// SIMATIC STEP 7 (V5.x) project TEST_212
// station: _S7H_BUSSYSTEM_CT
// station: P_ADR_BUS
// station: Hardware
// station: ESTACION_01

SYMBOL_TABLE
"Z 1"	C 1	COUNTER
"Z 2"	C 2	COUNTER
"Z 3"	C 3	COUNTER
"Z 4"	C 4	COUNTER
"Z 5"	C 5	COUNTER
"Z 6"	C 6	COUNTER
"Z 7"	C 7	COUNTER
"Z 8"	C 8	COUNTER
"Z 9"	C 9	COUNTER
"Z 10"	C 10	COUNTER
"Z 11"	C 11	COUNTER
"Z 12"	C 12	COUNTER
"Z 13"	C 13	COUNTER
"Z 14"	C 14	COUNTER
"Z 15"	C 15	COUNTER
"Z 16"	C 16	COUNTER
"Z 17"	C 17	COUNTER
"Z 18"	C 18	COUNTER
"Z 19"	C 19	COUNTER
"Z 20"	C 20	COUNTER
"Z 21"	C 21	COUNTER
"Z 22"	C 22	COUNTER
"Z 23"	C 23	COUNTER
"Z 24"	C 24	COUNTER
"Z 25"	C 25	COUNTER
"Z 26"	C 26	COUNTER
"Z 27"	C 27	COUNTER
"Z 28"	C 28	COUNTER
"Z 29"	C 29	COUNTER
"Z 30"	C 30	COUNTER
"Z 31"	C 31	COUNTER
"Z 32"	C 32	COUNTER
"Z 33"	C 33	COUNTER
"Z 34"	C 34	COUNTER
"Z 35"	C 35	COUNTER
"Z 36"	C 36	COUNTER
"Z 37"	C 37	COUNTER
"Z 38"	C 38	COUNTER
"Z 39"	C 39	COUNTER
"Z 40"	C 40	COUNTER
"Z 41"	C 41	COUNTER
"Z 42"	C 42	COUNTER
"Z 43"	C 43	COUNTER
"Z 44"	C 44	COUNTER
"Z 45"	C 45	COUNTER
"Z 46"	C 46	COUNTER
"Z 47"	C 47	COUNTER
"Z 48"	C 48	COUNTER
"Z 49"	C 49	COUNTER
"Z 50"	C 50	COUNTER
"Z 51"	C 51	COUNTER
"Z 52"	C 52	COUNTER
"Z 53"	C 53	COUNTER
"Z 54"	C 54	COUNTER
"Z 55"	C 55	COUNTER
"Z 56"	C 56	COUNTER
"Z 57"	C 57	COUNTER
"Z 58"	C 58	COUNTER
"Z 59"	C 59	COUNTER
"Z 60"	C 60	COUNTER
"Z 61"	C 61	COUNTER
"Z 62"	C 62	COUNTER
"Z 63"	C 63	COUNTER
"Z 64"	C 64	COUNTER
"Z 65"	C 65	COUNTER
"Z 66"	C 66	COUNTER
"Z 67"	C 67	COUNTER
"Z 68"	C 68	COUNTER
"Z 69"	C 69	COUNTER
"Z 70"	C 70	COUNTER
"Z 71"	C 71	COUNTER
"Z 72"	C 72	COUNTER
"Z 73"	C 73	COUNTER
"Z 74"	C 74	COUNTER
"Z 75"	C 75	COUNTER
"Z 76"	C 76	COUNTER
"Z 77"	C 77	COUNTER
"Z 78"	C 78	COUNTER
"Z 79"	C 79	COUNTER
"Z 80"	C 80	COUNTER
"Z 81"	C 81	COUNTER
"Z 82"	C 82	COUNTER
"Z 83"	C 83	COUNTER
"Z 84"	C 84	COUNTER
"Z 85"	C 85	COUNTER
"Z 86"	C 86	COUNTER
"Z 87"	C 87	COUNTER
"Z 88"	C 88	COUNTER
"Z 89"	C 89	COUNTER
"Z 90"	C 90	COUNTER
"Z 91"	C 91	COUNTER
"Z 92"	C 92	COUNTER
"Z 93"	C 93	COUNTER
"Z 94"	C 94	COUNTER
"Z 95"	C 95	COUNTER
"Z 96"	C 96	COUNTER
"Z 97"	C 97	COUNTER
"Z 98"	C 98	COUNTER
"Z 99"	C 99	COUNTER
"Z 100"	C 100	COUNTER	// CONTADOR DE MINUTOS ( ALARMA  )
"Z 101"	C 101	COUNTER	// CONTADOR DE HORAS ( ALARMA  )
"Z 102"	C 102	COUNTER	// CONTADOR DE SEGUNDOS ( RELOJ  )
"Z 103"	C 103	COUNTER	// CONTADOR DE MINUTOS ( RELOJ )
"Z 104"	C 104	COUNTER	// CONTADOR DE HORAS ( RELOJ  )
"Z 105"	C 105	COUNTER	// CONTADOR DE RELOJ ( RELOJ DE 24 HORAS )
"Z 106"	C 106	COUNTER
"Z 107"	C 107	COUNTER
"Z 108"	C 108	COUNTER
"Z 109"	C 109	COUNTER
"Z 110"	C 110	COUNTER	// CONTADOR DE MINUTOS - AJUSTE DE ALARMAS
"Z 111"	C 111	COUNTER
"Z 112"	C 112	COUNTER
"Z 113"	C 113	COUNTER
"Z 114"	C 114	COUNTER
"Z 115"	C 115	COUNTER
"Z 116"	C 116	COUNTER
"Z 117"	C 117	COUNTER
"Z 118"	C 118	COUNTER
"Z 119"	C 119	COUNTER	// CONTADOR DE PERSONAS
"Z 120"	C 120	COUNTER	// CONTADOR ASCENDENTE / DESCENDENTE
"Z 121"	C 121	COUNTER	// CONTADOR ASCENDENTE
"Z 122"	C 122	COUNTER	// CONTADOR DESCENDENTE
"Z 123"	C 123	COUNTER
"Z 124"	C 124	COUNTER
"Z 125"	C 125	COUNTER
"Z 126"	C 126	COUNTER
"Z 127"	C 127	COUNTER	// CONTADOR DE IMPULSOS
"Z 128"	C 128	COUNTER
"Z 129"	C 129	COUNTER
"Z 130"	C 130	COUNTER
"Z 131"	C 131	COUNTER
"Z 132"	C 132	COUNTER
"Z 133"	C 133	COUNTER
"Z 134"	C 134	COUNTER
"Z 135"	C 135	COUNTER
"Z 136"	C 136	COUNTER
"Z 137"	C 137	COUNTER
"Z 138"	C 138	COUNTER
"Z 139"	C 139	COUNTER
"Z 140"	C 140	COUNTER
"Z 141"	C 141	COUNTER
"Z 142"	C 142	COUNTER
"Z 143"	C 143	COUNTER
"Z 144"	C 144	COUNTER
"Z 145"	C 145	COUNTER
"Z 146"	C 146	COUNTER
"Z 147"	C 147	COUNTER
"Z 148"	C 148	COUNTER
"Z 149"	C 149	COUNTER
"Z 150"	C 150	COUNTER
"Z 151"	C 151	COUNTER
"Z 152"	C 152	COUNTER
"Z 153"	C 153	COUNTER
"Z 154"	C 154	COUNTER
"Z 155"	C 155	COUNTER
"Z 156"	C 156	COUNTER
"Z 157"	C 157	COUNTER
"Z 158"	C 158	COUNTER
"Z 159"	C 159	COUNTER
"Z 160"	C 160	COUNTER
"Z 161"	C 161	COUNTER
"Z 162"	C 162	COUNTER
"Z 163"	C 163	COUNTER
"Z 164"	C 164	COUNTER
"Z 165"	C 165	COUNTER
"Z 166"	C 166	COUNTER
"Z 167"	C 167	COUNTER
"Z 168"	C 168	COUNTER
"Z 169"	C 169	COUNTER
"Z 170"	C 170	COUNTER
"Z 171"	C 171	COUNTER
"Z 172"	C 172	COUNTER
"Z 173"	C 173	COUNTER
"Z 174"	C 174	COUNTER
"Z 175"	C 175	COUNTER
"Z 176"	C 176	COUNTER
"Z 177"	C 177	COUNTER
"Z 178"	C 178	COUNTER
"Z 179"	C 179	COUNTER
"Z 180"	C 180	COUNTER
"Z 181"	C 181	COUNTER
"Z 182"	C 182	COUNTER
"Z 183"	C 183	COUNTER
"Z 184"	C 184	COUNTER
"Z 185"	C 185	COUNTER
"Z 186"	C 186	COUNTER
"Z 187"	C 187	COUNTER
"Z 188"	C 188	COUNTER
"Z 189"	C 189	COUNTER
"Z 190"	C 190	COUNTER
"Z 191"	C 191	COUNTER
"Z 192"	C 192	COUNTER
"Z 193"	C 193	COUNTER
"Z 194"	C 194	COUNTER
"Z 195"	C 195	COUNTER
"Z 196"	C 196	COUNTER
"Z 197"	C 197	COUNTER
"Z 198"	C 198	COUNTER
"Z 199"	C 199	COUNTER
"Z 200"	C 200	COUNTER
"Z 201"	C 201	COUNTER
"Z 202"	C 202	COUNTER
"Z 203"	C 203	COUNTER
"Z 204"	C 204	COUNTER
"Z 205"	C 205	COUNTER
"Z 206"	C 206	COUNTER
"Z 207"	C 207	COUNTER
"Z 208"	C 208	COUNTER
"Z 209"	C 209	COUNTER
"Z 210"	C 210	COUNTER
"Z 211"	C 211	COUNTER
"Z 212"	C 212	COUNTER
"Z 213"	C 213	COUNTER
"Z 214"	C 214	COUNTER
"Z 215"	C 215	COUNTER
"Z 216"	C 216	COUNTER
"Z 217"	C 217	COUNTER
"Z 218"	C 218	COUNTER
"Z 219"	C 219	COUNTER
"Z 220"	C 220	COUNTER
"Z 221"	C 221	COUNTER
"Z 222"	C 222	COUNTER
"Z 223"	C 223	COUNTER
"Z 224"	C 224	COUNTER
"Z 225"	C 225	COUNTER
"Z 226"	C 226	COUNTER
"Z 227"	C 227	COUNTER
"Z 228"	C 228	COUNTER
"Z 229"	C 229	COUNTER
"Z 230"	C 230	COUNTER
"Z 231"	C 231	COUNTER
"Z 232"	C 232	COUNTER
"Z 233"	C 233	COUNTER
"Z 234"	C 234	COUNTER
"Z 235"	C 235	COUNTER
"Z 236"	C 236	COUNTER
"Z 237"	C 237	COUNTER
"Z 238"	C 238	COUNTER
"Z 239"	C 239	COUNTER
"Z 240"	C 240	COUNTER
"Z 241"	C 241	COUNTER
"Z 242"	C 242	COUNTER
"Z 243"	C 243	COUNTER
"Z 244"	C 244	COUNTER
"Z 245"	C 245	COUNTER
"Z 246"	C 246	COUNTER
"Z 247"	C 247	COUNTER
"Z 248"	C 248	COUNTER
"Z 249"	C 249	COUNTER
"Z 250"	C 250	COUNTER
"Z 251"	C 251	COUNTER
"Z 252"	C 252	COUNTER
"Z 253"	C 253	COUNTER
"Z 254"	C 254	COUNTER
"Z 255"	C 255	COUNTER
"Z 256"	C 256	COUNTER
"DB 126"	DB 126	FB 126	// InstanzDB PNIODiag
"DB 127"	DB 127	DB 127	// InstanzDB STATDiag
"DB 208"	DB 208	DB 208	// DATOS GENERALES - TAK SIGNALE
"DB 228"	DB 228	DB 228	// SALVADO DE MARCAS OB35
"PNIODiag"	FB 126	FB 126	// Profibus/DP und Profinet/IO-Diagnose
"STATDiag"	FB 127	FB 127	// Zweitbaustein (PNIODiag)
"TE-M/V"	FC 10	FC 10	// FUNCIONAMIENTO DE ACCIONAMIENTO ( MOTOR / VALVULA )
"TE-SS"	FC 11	FC 11	// FUNCIONAMIENTO DE ACCIONAMIENTO ( VALVULA MOTORIZADA )
"TE-REK"	FC 12	FC 12	// FUNCIONAMIENTO DE ACCIONAMIENTO ( VALVULA DE CONTROL )
"TE-TS"	FC 13	FC 13	// FUNCIONAMIENTO DE ACCIONAMIENTO ( CONTROL PARCIAL )
"TE-VW3/3"	FC 14	FC 14	// FUNCIONAMIENTO DE ACCIONAMIENTO ( PRESELECCION 1 )
"TE-KO"	FC 15	FC 15	// FUNCIONAMIENTO DE CONTROL DE PASOS ( SECUENCIALES )
"TE-VW2/2"	FC 16	FC 16	// FUNCIONAMIENTO DE ACCIONAMIENTO ( PRESELECCION 1 )
"TE-VW2/1"	FC 17	FC 17	// FUNCIONAMIENTO DE ACCIONAMIENTO ( PRESELECCION 1 )
"TE_READ_RTM"	FC 18	FC 18	// TIEMPO DE FUNCIONAMIENTO DE UN ACCIONAMIENTO
"TE-WL ( PEA )"	FC 20	FC 20	// SENTRON WL ( IMAGEN DE PROCESO DE SALIDAS )
"TE-WL ( PEE )"	FC 25	FC 25	// SENTRON WL ( IMAGEN DE PROCESO DE ENTRADAS )
"TE-TAK"	FC 29	FC 29	// FUNCION DE GENERACION DE IMPULSOS
"TE-GRENZ"	FC 36	FC 36	// FUNCION DE LIMITE DE ALARMAS
"TE-RETTEN"	FC 38	FC 38	// SALVADO DE MARCAS DE TRABAJO
"TE-LADEN"	FC 39	FC 39	// CARGA DE MARCAS DE TRABAJO
"TE-SCHALTER"	FC 49	FC 49	// ANALOGSCHALTER - FUNKTION
"G7_STD_3"	FC 72	FC 72	// CONTROL DE OPERACION DE SECUENCIAS - GRAPH 7
"TE-ANEI"	FC 78	FC 78	// FUNCION DE LECTURA ANALOGICA
"TE-ANAU"	FC 79	FC 79	// FUNCION DE SALIDA ANALOGICA
"FC 110"	FC 110	FC 110	// FUNCIONES BASICAS
"FC 111"	FC 111	FC 111	// OPERACIONES LOGICAS BINARIAS
"FC 112"	FC 112	FC 112	// FUNCIONES DE MEMORIA
"FC 113"	FC 113	FC 113	// TEMPORIZADORES
"FC 114"	FC 114	FC 114	// CONTADORES
"FC 120"	FC 120	FC 120	// EJEMPLOS DE LAS FUNCIONES BINARIAS
"FC 121"	FC 121	FC 121	// SUPERVISION DE VENTILADORES
"FC 122"	FC 122	FC 122	// SUPERVISION DE FRECUENCIAS
"FC 123"	FC 123	FC 123	// CONTADOR DE PERSONAL
"FC 124"	FC 124	FC 124	// GENERADOR DE IMPULSOS
"FC 125"	FC 125	FC 125	// SEMAFORO
"FC 130"	FC 130	FC 130	// DIAGRAMAS ELECTRICOS
"FC 131"	FC 131	FC 131	// EJERCICIO No. 1 - CIRCUITO DE ENCLAVAMIENTO
"FC 132"	FC 132	FC 132	// EJERCICIO No. 2 - CIRCUITO DE TEMPORIZACION
"FC 133"	FC 133	FC 133	// EJERCICIO No. 3 - INVERSION DE GIRO
"FC 134"	FC 134	FC 134	// EJERCICIO No. 4 - ARRANQUE ESTRELLA - TRIANGULO
"FC 135"	FC 135	FC 135	// EJERCICIO No. 5 - INVERSION DE GIRO CON ARRANQUE ESTRELLA  - TRIANGULO
"FC 136"	FC 136	FC 136	// EJERCICIO No. 6 - CONEXION DAHLANDER
"FC 137"	FC 137	FC 137	// EJERCICIO No. 7 - MONTACARGAS
"FC 140"	FC 140	FC 140	// EJERCICIOS DE FUNCIONES BINARIAS
"FC 141"	FC 141	FC 141	// EJERCICIO No. 1 - SEMAFORO
"FC 142"	FC 142	FC 142	// EJERCICIO No. 2 - RELOJ DESPERTADOR
"FC 143"	FC 143	FC 143	// EJERCICIO No. 3 - PANEL DE ALARMAS
"FC 144"	FC 144	FC 144	// EJERCICIO No. 4 - ARRANQUE Y PARO DE MOTORES
"FC 145"	FC 145	FC 145	// EJERCICIO No. 5 - ELEVADOR
"FC 150"	FC 150	FC 150
"FC 151"	FC 151	FC 151
"FC 160"	FC 160	FC 160	// DIAGRAMAS ELECTRONEUMATICOS
"FC 161"	FC 161	FC 161	// EJERCICIO No. 1 -
"FC 162"	FC 162	FC 162	// EJERCICIO No. 2 -
"FC 163"	FC 163	FC 163	// EJERCICIO No. 3 -
"FC 164"	FC 164	FC 164	// EJERCICIO No. 4 -
"FC 165"	FC 165	FC 165	// EJERCICIO No. 5 -
"FC 166"	FC 166	FC 166	// EJERCICIO No. 6 -
"FC 167"	FC 167	FC 167	// EJERCICIO No. 7 -
"FC 240"	FC 240	FC 240	// INDICACION DE ESTADO - PANEL DE OPERACION
"FC 248"	FC 248	FC 248	// INDICACION DE CONTACTORES
"FC 249"	FC 249	FC 249	// INDICACION DE SELECTORES
"FC 250"	FC 250	FC 250	// SIMULACION DE RETROAVISOS
"FC 251"	FC 251	FC 251	// SIMULACION DE RETROAVISOS # 1
"FC 252"	FC 252	FC 252	// SIMULACION DE RETROAVISOS # 2
"FC 253"	FC 253	FC 253	// SIMULACION DE RETROAVISOS # 3
"FC 254"	FC 254	FC 254	// SIMULACION DE RETROAVISOS # 4
"FC 255"	FC 255	FC 255	// SIMULACION DE RETROAVISOS # 5
"FC 256"	FC 256	FC 256	// SIMULACION DE RETROAVISOS # 6
"FC 257"	FC 257	FC 257	// SIMULACION DE RETROAVISOS # 7
"1S2"	I 0.0	BOOL	// BOTON PULSADOR DE ARRANQUE # 1
"2S2"	I 0.1	BOOL	// BOTON PULSADOR DE ARRANQUE # 2
"3S2"	I 0.2	BOOL	// BOTON PULSADOR DE ARRANQUE # 3
"4S2"	I 0.3	BOOL	// BOTON PULSADOR DE ARRANQUE # 4
"5S2"	I 0.4	BOOL	// BOTON PULSADOR DE ARRANQUE # 5
"6S2"	I 0.5	BOOL	// BOTON PULSADOR DE ARRANQUE # 6
"7S2"	I 0.6	BOOL	// BOTON PULSADOR DE ARRANQUE # 7
"8S2"	I 0.7	BOOL	// BOTON PULSADOR DE ARRANQUE # 8
"1S3"	I 1.0	BOOL	// BOTON PULSADOR DE PARO # 1
"2S3"	I 1.1	BOOL	// BOTON PULSADOR DE PARO # 2
"3S3"	I 1.2	BOOL	// BOTON PULSADOR DE PARO # 3
"4S3"	I 1.3	BOOL	// BOTON PULSADOR DE PARO # 4
"5S3"	I 1.4	BOOL	// BOTON PULSADOR DE PARO # 5
"6S3"	I 1.5	BOOL	// BOTON PULSADOR DE PARO # 6
"7S3"	I 1.6	BOOL	// BOTON PULSADOR DE PARO # 7
"8S3"	I 1.7	BOOL	// BOTON PULSADOR DE PARO # 8
"1FR1"	I 2.0	BOOL	// DISPOSITIVO DE PROTECCION ( POR UMBRAL DE INTENSIDAD ) # 1
"2FR1"	I 2.1	BOOL	// DISPOSITIVO DE PROTECCION ( POR UMBRAL DE INTENSIDAD ) # 2
"3FR1"	I 2.2	BOOL	// DISPOSITIVO DE PROTECCION ( POR UMBRAL DE INTENSIDAD ) # 3
"4FR1"	I 2.3	BOOL	// DISPOSITIVO DE PROTECCION ( POR UMBRAL DE INTENSIDAD ) # 4
"5FR1"	I 2.4	BOOL	// DISPOSITIVO DE PROTECCION ( POR UMBRAL DE INTENSIDAD ) # 5
"6FR1"	I 2.5	BOOL	// DISPOSITIVO DE PROTECCION ( POR UMBRAL DE INTENSIDAD ) # 6
"7FR1"	I 2.6	BOOL	// DISPOSITIVO DE PROTECCION ( POR UMBRAL DE INTENSIDAD ) # 7
"8FR1"	I 2.7	BOOL	// DISPOSITIVO DE PROTECCION ( POR UMBRAL DE INTENSIDAD ) # 8
"E 3.0"	I 3.0	BOOL
"E 3.1"	I 3.1	BOOL
"E 3.2"	I 3.2	BOOL
"E 3.3"	I 3.3	BOOL
"E 3.4"	I 3.4	BOOL
"E 3.5"	I 3.5	BOOL
"E 3.6"	I 3.6	BOOL
"E 3.7"	I 3.7	BOOL
"5KM1_12"	I 4.0	BOOL	// CONTACTOR PRINCIPAL - 5KM1 ( DESCONECTADO )
"5KM1_14"	I 4.1	BOOL	// CONTACTOR PRINCIPAL - 5KM1 ( CONECTADO )
"5KM2_12"	I 4.2	BOOL	// CONTACTOR PRINCIPAL - 5KM2 ( DESCONECTADO )
"5KM2_14"	I 4.3	BOOL	// CONTACTOR PRINCIPAL - 5KM2 ( CONECTADO )
"5KM3_12"	I 4.4	BOOL	// CONTACTOR PRINCIPAL - 5KM3 ( DESCONECTADO )
"5KM3_14"	I 4.5	BOOL	// CONTACTOR PRINCIPAL - 5KM3 ( CONECTADO )
"5KM4_12"	I 4.6	BOOL	// CONTACTOR PRINCIPAL - 5KM4 ( DESCONECTADO )
"5KM4_14"	I 4.7	BOOL	// CONTACTOR PRINCIPAL - 5KM4 ( CONECTADO )
"6KM1_12"	I 5.0	BOOL	// CONTACTOR PRINCIPAL - 6KM1 ( DESCONECTADO )
"6KM1_14"	I 5.1	BOOL	// CONTACTOR PRINCIPAL - 6KM1 ( CONECTADO )
"6KM2_12"	I 5.2	BOOL	// CONTACTOR PRINCIPAL - 6KM2 ( DESCONECTADO )
"6KM2_14"	I 5.3	BOOL	// CONTACTOR PRINCIPAL - 6KM2 ( CONECTADO )
"6KM3_12"	I 5.4	BOOL	// CONTACTOR PRINCIPAL - 6KM3 ( DESCONECTADO )
"6KM3_14"	I 5.5	BOOL	// CONTACTOR PRINCIPAL - 6KM3 ( CONECTADO )
"E 5.6"	I 5.6	BOOL
"E 5.7"	I 5.7	BOOL
"1KM1_12"	I 6.0	BOOL	// CONTACTOR PRINCIPAL - 1KM1 ( DESCONECTADO )
"1KM1_14"	I 6.1	BOOL	// CONTACTOR PRINCIPAL - 1KM1 ( CONECTADO )
"2KM1_12"	I 6.2	BOOL	// CONTACTOR PRINCIPAL - 2KM1 ( DESCONECTADO )
"2KM1_14"	I 6.3	BOOL	// CONTACTOR PRINCIPAL - 2KM1 ( CONECTADO )
"2KM2_12"	I 6.4	BOOL	// CONTACTOR PRINCIPAL - 2KM2 ( DESCONECTADO )
"2KM2_14"	I 6.5	BOOL	// CONTACTOR PRINCIPAL - 2KM2 ( CONECTADO )
"E 6.6"	I 6.6	BOOL
"E 6.7"	I 6.7	BOOL
"BE4"	I 8.0	BOOL	// TRANSPORTADOR - SENSOR LB
"S1"	I 8.1	BOOL	// TRANSPORTADOR - BOTON PULSADOR T_BAY1
"S2"	I 8.2	BOOL	// TRANSPORTADOR - BOTON PULSADOR T_BAY2
"S3"	I 8.3	BOOL	// TRANSPORTADOR - BOTON PULSADOR T_BAY3
"S4"	I 8.4	BOOL	// TRANSPORTADOR - BOTON PULSADOR T_BAY-LB
"BE1"	I 8.5	BOOL	// TRANSPORTADOR - SENSOR BAY1
"BE2"	I 8.6	BOOL	// TRANSPORTADOR - SENSOR BAY2
"BE3"	I 8.7	BOOL	// TRANSPORTADOR - SENSOR BAY3
"3KM1_12"	I 12.0	BOOL	// CONTACTOR PRINCIPAL - 3KM1 ( DESCONECTADO )
"3KM1_14"	I 12.1	BOOL	// CONTACTOR PRINCIPAL - 3KM1 ( CONECTADO )
"3KM2_12"	I 12.2	BOOL	// CONTACTOR PRINCIPAL - 3KM2 ( DESCONECTADO )
"3KM2_14"	I 12.3	BOOL	// CONTACTOR PRINCIPAL - 3KM2 ( CONECTADO )
"E 12.4"	I 12.4	BOOL
"E 12.5"	I 12.5	BOOL
"E 12.6"	I 12.6	BOOL
"E 12.7"	I 12.7	BOOL
"4KM1_12"	I 13.0	BOOL	// CONTACTOR PRINCIPAL - 4KM1 ( DESCONECTADO )
"4KM1_14"	I 13.1	BOOL	// CONTACTOR PRINCIPAL - 4KM1 ( CONECTADO )
"4KM2_12"	I 13.2	BOOL	// CONTACTOR PRINCIPAL - 4KM2 ( DESCONECTADO )
"4KM2_14"	I 13.3	BOOL	// CONTACTOR PRINCIPAL - 4KM2 ( CONECTADO )
"4KM3_12"	I 13.4	BOOL	// CONTACTOR PRINCIPAL - 4KM3 ( DESCONECTADO )
"4KM3_14"	I 13.5	BOOL	// CONTACTOR PRINCIPAL - 4KM3 ( CONECTADO )
"E 13.6"	I 13.6	BOOL
"E 13.7"	I 13.7	BOOL
"E 14.0"	I 14.0	BOOL
"E 14.1"	I 14.1	BOOL
"E 14.2"	I 14.2	BOOL
"E 14.3"	I 14.3	BOOL
"E 14.4"	I 14.4	BOOL
"E 14.5"	I 14.5	BOOL
"E 14.6"	I 14.6	BOOL
"E 14.7"	I 14.7	BOOL
"E 15.0"	I 15.0	BOOL
"E 15.1"	I 15.1	BOOL
"E 15.2"	I 15.2	BOOL
"E 15.3"	I 15.3	BOOL
"E 15.4"	I 15.4	BOOL
"E 15.5"	I 15.5	BOOL
"E 15.6"	I 15.6	BOOL
"E 15.7"	I 15.7	BOOL
"7KM1_12"	I 16.0	BOOL	// CONTACTOR DE VELOCIDAD LENTA ( DESCONECTADO )
"7KM1_14"	I 16.1	BOOL
"7KM2_12"	I 16.2	BOOL	// CONTACTOR DE VELOCIDAD RAPIDA ( DESCONECTADO )
"7KM2_!4"	I 16.3	BOOL
"7KM3_12"	I 16.4	BOOL	// CONTACTOR DE VELOCIDAD RAPIDA ( DESCONECTADO )
"7KM3_14"	I 16.5	BOOL	// CONTACTOR DE VELOCIDAD RAPIDA ( CONECTADO )
"7QS10"	I 16.6	BOOL	// DETECTOR DE PLANTA BAJA
"7QS20"	I 16.7	BOOL	// DETECTOR PRIMER PISO
"7KM10_12"	I 17.0	BOOL	// CONTACTOR DE BAJADA ( DESCONECTADO )
"7KM10_14"	I 17.1	BOOL	// CONTACTOR DE BAJADA ( CONECTADO )
"7KM20_12"	I 17.2	BOOL	// CONTACTOR DE SUBIDA ( DESCONECTADO )
"7KM20_14"	I 17.3	BOOL	// CONTACTOR DE SUBIDA ( CONECTADO )
"7SB1"	I 17.4	BOOL	// COMANDO DE LLAMADA A PLANTA BAJA
"7SB2"	I 17.5	BOOL	// COMANDO DE LLAMADA A PRIMER PISO
"7SB3"	I 17.6	BOOL	// COMANDO DE PARO
"1S1A"	I 124.0	BOOL	// POSICION LOCAL - SELECTOR # 1
"1S1B"	I 124.1	BOOL	// POSICION REMOTO - SELECTOR # 1
"2S1A"	I 124.2	BOOL	// POSICION LOCAL - SELECTOR # 2
"2S1B"	I 124.3	BOOL	// POSICION REMOTO - SELECTOR # 2
"3S1A"	I 124.4	BOOL	// POSICION LOCAL - SELECTOR # 3
"3S1B"	I 124.5	BOOL	// POSICION REMOTO - SELECTOR # 3
"4S1A"	I 124.6	BOOL	// POSICION LOCAL - SELECTOR # 4
"4S1B"	I 124.7	BOOL	// POSICION REMOTO - SELECTOR # 4
"5S1A"	I 125.0	BOOL	// POSICION LOCAL - SELECTOR # 5
"5S1B"	I 125.1	BOOL	// POSICION REMOTO - SELECTOR # 5
"6S1A"	I 125.2	BOOL	// POSICION LOCAL - SELECTOR # 6
"6S1B"	I 125.3	BOOL	// POSICION REMOTO - SELECTOR # 6
"7S1A"	I 125.4	BOOL	// POSICION LOCAL - SELECTOR # 7
"7S1B"	I 125.5	BOOL	// POSICION REMOTO - SELECTOR # 7
"8S1A"	I 125.6	BOOL	// POSICION LOCAL - SELECTOR # 8
"8S1B"	I 125.7	BOOL	// POSICION REMOTO - SELECTOR # 8
"´0´"	M 0.0	BOOL	// CERO LOGICO
"´1´"	M 0.1	BOOL	// UNO LOGICO
"M 0.2"	M 0.2	BOOL
"M 0.3"	M 0.3	BOOL
"M 0.4"	M 0.4	BOOL
"M 0.5"	M 0.5	BOOL
"M 0.6"	M 0.6	BOOL	// MARCA DE INICIO - PROGRAMA DE TIEMPO ( 100 ms )
"M 0.7"	M 0.7	BOOL	// MARCA DE INICIO - EJECUCION CICLICA DE PROGRAMA
"M 1.0"	M 1.0	BOOL
"M 1.1"	M 1.1	BOOL
"M 1.2"	M 1.2	BOOL	// FLANCO 0.5 Seg.
"M 1.3"	M 1.3	BOOL	// FLANCO 1.0 Seg.
"M 1.4"	M 1.4	BOOL	// FLANCO 2.0 Seg.
"M 1.5"	M 1.5	BOOL	// PULSOS 0.5 Seg.
"M 1.6"	M 1.6	BOOL	// PULSOS 1.0 Seg.
"M 1.7"	M 1.7	BOOL	// PULSOS 2.0 Seg.
"M 2.0"	M 2.0	BOOL
"M 2.1"	M 2.1	BOOL
"M 2.2"	M 2.2	BOOL
"M 2.3"	M 2.3	BOOL
"M 2.4"	M 2.4	BOOL
"M 2.5"	M 2.5	BOOL
"M 2.6"	M 2.6	BOOL
"M 2.7"	M 2.7	BOOL
"M 3.0"	M 3.0	BOOL
"M 3.1"	M 3.1	BOOL
"M 3.2"	M 3.2	BOOL
"M 3.3"	M 3.3	BOOL
"M 3.4"	M 3.4	BOOL
"M 3.5"	M 3.5	BOOL
"M 3.6"	M 3.6	BOOL
"M 3.7"	M 3.7	BOOL
"M 4.0"	M 4.0	BOOL
"M 4.1"	M 4.1	BOOL
"M 4.2"	M 4.2	BOOL
"M 4.3"	M 4.3	BOOL
"M 4.4"	M 4.4	BOOL
"M 4.5"	M 4.5	BOOL
"M 4.6"	M 4.6	BOOL
"M 4.7"	M 4.7	BOOL
"M 5.0"	M 5.0	BOOL
"M 5.1"	M 5.1	BOOL
"M 5.2"	M 5.2	BOOL
"M 5.3"	M 5.3	BOOL
"M 5.4"	M 5.4	BOOL
"M 5.5"	M 5.5	BOOL
"M 5.6"	M 5.6	BOOL
"M 5.7"	M 5.7	BOOL
"M 6.0"	M 6.0	BOOL
"M 6.1"	M 6.1	BOOL
"M 6.2"	M 6.2	BOOL
"M 6.3"	M 6.3	BOOL
"M 6.4"	M 6.4	BOOL
"M 6.5"	M 6.5	BOOL
"M 6.6"	M 6.6	BOOL
"M 6.7"	M 6.7	BOOL
"M 7.0"	M 7.0	BOOL
"M 7.1"	M 7.1	BOOL
"M 7.2"	M 7.2	BOOL
"M 7.3"	M 7.3	BOOL
"M 7.4"	M 7.4	BOOL
"M 7.5"	M 7.5	BOOL
"M 7.6"	M 7.6	BOOL
"M 7.7"	M 7.7	BOOL
"M 8.0"	M 8.0	BOOL
"M 8.1"	M 8.1	BOOL
"M 8.2"	M 8.2	BOOL
"M 8.3"	M 8.3	BOOL
"M 8.4"	M 8.4	BOOL
"M 8.5"	M 8.5	BOOL
"M 8.6"	M 8.6	BOOL
"M 8.7"	M 8.7	BOOL
"M 9.0"	M 9.0	BOOL
"M 9.1"	M 9.1	BOOL
"M 9.2"	M 9.2	BOOL
"M 9.3"	M 9.3	BOOL
"M 9.4"	M 9.4	BOOL
"M 9.5"	M 9.5	BOOL
"M 9.6"	M 9.6	BOOL
"M 9.7"	M 9.7	BOOL
"M 10.0"	M 10.0	BOOL	// PANEL DE OPERACION ( COMANDO DE ARRANQUE )
"M 10.7"	M 10.7	BOOL	// MARCA AUXILIAR - COMANDO DE ARRANQUE
"M 11.0"	M 11.0	BOOL	// PANEL DE OPERACION ( BOTON PULSADOR DE  ARRANQUE # 1 )
"M 11.1"	M 11.1	BOOL	// PANEL DE OPERACION ( BOTON PULSADOR DE  ARRANQUE # 2 )
"M 11.2"	M 11.2	BOOL	// PANEL DE OPERACION ( BOTON PULSADOR DE PARO )
"M 11.3"	M 11.3	BOOL
"M 11.4"	M 11.4	BOOL	// MARCA AUXILIAR - SIMULACION DE RETROAVISOS # 1
"M 11.5"	M 11.5	BOOL	// MARCA AUXILIAR - COMANDO DE PARO
"M 11.6"	M 11.6	BOOL	// MARCA AUXILIAR - COMANDO DE ARRANQUE # 2
"M 11.7"	M 11.7	BOOL	// MARCA AUXILIAR - COMANDO DE ARRANQUE # 1
"M 12.0"	M 12.0	BOOL	// PANEL DE OPERACION ( BOTON PULSADOR DE  ARRANQUE # 1 )
"M 12.1"	M 12.1	BOOL	// PANEL DE OPERACION ( BOTON PULSADOR DE  ARRANQUE # 2 )
"M 12.2"	M 12.2	BOOL	// PANEL DE OPERACION ( BOTON PULSADOR DE PARO )
"M 12.3"	M 12.3	BOOL	// MARCA AUXILIAR - SIMULACION DE RETROAVISOS # 2
"M 12.4"	M 12.4	BOOL	// MARCA AUXILIAR - SIMULACION DE RETROAVISOS # 1
"M 12.5"	M 12.5	BOOL	// MARCA AUXILIAR - COMANDO DE PARO
"M 12.6"	M 12.6	BOOL	// MARCA AUXILIAR - COMANDO DE ARRANQUE # 2
"M 12.7"	M 12.7	BOOL	// MARCA AUXILIAR - COMANDO DE ARRANQUE # 1
"M 13.0"	M 13.0	BOOL	// PANEL DE OPERACION ( BOTON PULSADOR DE  ARRANQUE # 1 )
"M 13.1"	M 13.1	BOOL	// PANEL DE OPERACION ( BOTON PULSADOR DE  ARRANQUE # 2 )
"M 13.2"	M 13.2	BOOL	// PANEL DE OPERACION ( BOTON PULSADOR DE PARO )
"M 13.3"	M 13.3	BOOL	// MARCA AUXILIAR - SIMULACION DE RETROAVISOS # 2
"M 13.4"	M 13.4	BOOL	// MARCA AUXILIAR - SIMULACION DE RETROAVISOS # 1
"M 13.5"	M 13.5	BOOL	// MARCA AUXILIAR - COMANDO DE PARO
"M 13.6"	M 13.6	BOOL	// MARCA AUXILIAR - COMANDO DE ARRANQUE # 2
"M 13.7"	M 13.7	BOOL	// MARCA AUXILIAR - COMANDO DE ARRANQUE # 1
"M 14.0"	M 14.0	BOOL	// PANEL DE OPERACION ( BOTON PULSADOR DE  ARRANQUE # 1 )
"M 14.1"	M 14.1	BOOL	// PANEL DE OPERACION ( BOTON PULSADOR DE  ARRANQUE # 2 )
"M 14.2"	M 14.2	BOOL	// PANEL DE OPERACION ( BOTON PULSADOR DE PARO )
"M 14.3"	M 14.3	BOOL	// MARCA AUXILIAR - SIMULACION DE RETROAVISOS # 2
"M 14.4"	M 14.4	BOOL	// MARCA AUXILIAR - SIMULACION DE RETROAVISOS # 1
"M 14.5"	M 14.5	BOOL	// MARCA AUXILIAR - COMANDO DE PARO
"M 14.6"	M 14.6	BOOL	// MARCA AUXILIAR - COMANDO DE ARRANQUE # 2
"M 14.7"	M 14.7	BOOL	// MARCA AUXILIAR - COMANDO DE ARRANQUE # 1
"M 15.0"	M 15.0	BOOL	// PANEL DE OPERACION ( BOTON PULSADOR DE  ARRANQUE # 1 )
"M 15.1"	M 15.1	BOOL	// PANEL DE OPERACION ( BOTON PULSADOR DE  ARRANQUE # 2 )
"M 15.2"	M 15.2	BOOL	// PANEL DE OPERACION ( BOTON PULSADOR DE PARO )
"M 15.3"	M 15.3	BOOL	// MARCA AUXILIAR - SIMULACION DE RETROAVISOS # 2
"M 15.4"	M 15.4	BOOL	// MARCA AUXILIAR - SIMULACION DE RETROAVISOS # 1
"M 15.5"	M 15.5	BOOL	// MARCA AUXILIAR - COMANDO DE PARO
"M 15.6"	M 15.6	BOOL	// MARCA AUXILIAR - COMANDO DE ARRANQUE # 2
"M 15.7"	M 15.7	BOOL	// MARCA AUXILIAR - COMANDO DE ARRANQUE # 1
"M 16.0"	M 16.0	BOOL	// PANEL DE OPERACION ( BOTON PULSADOR DE  ARRANQUE # 1 )
"M 16.1"	M 16.1	BOOL	// PANEL DE OPERACION ( BOTON PULSADOR DE  ARRANQUE # 2 )
"M 16.2"	M 16.2	BOOL	// PANEL DE OPERACION ( BOTON PULSADOR DE PARO )
"M 16.3"	M 16.3	BOOL	// MARCA AUXILIAR - SIMULACION DE RETROAVISOS # 2
"M 16.4"	M 16.4	BOOL	// MARCA AUXILIAR - SIMULACION DE RETROAVISOS # 1
"M 16.5"	M 16.5	BOOL	// MARCA AUXILIAR - COMANDO DE PARO
"M 16.6"	M 16.6	BOOL	// MARCA AUXILIAR - COMANDO DE ARRANQUE # 2
"M 16.7"	M 16.7	BOOL	// MARCA AUXILIAR - COMANDO DE ARRANQUE # 1
"M 17.0"	M 17.0	BOOL	// PANEL DE OPERACION ( COMANDO - LLAMADA A PLANTA BAJA  )
"M 17.1"	M 17.1	BOOL	// PANEL DE OPERACION ( COMANDO - LLAMADA A PRIMER PISO  )
"M 17.2"	M 17.2	BOOL	// PANEL DE OPERACION ( COMANDO DE PARO - MONTACARGAS )
"M 17.3"	M 17.3	BOOL	// MARCA AUXILIAR - SIMULACION DE RETROAVISOS # 2
"M 17.4"	M 17.4	BOOL	// MARCA AUXILIAR - SIMULACION DE RETROAVISOS # 1
"M 17.5"	M 17.5	BOOL	// MARCA AUXILIAR - COMANDO DE PARO
"M 17.6"	M 17.6	BOOL	// MARCA AUXILIAR - COMANDO DE ARRANQUE # 2
"M 17.7"	M 17.7	BOOL	// MARCA AUXILIAR - COMANDO DE ARRANQUE # 1
"M 18.0"	M 18.0	BOOL
"M 18.1"	M 18.1	BOOL
"M 18.2"	M 18.2	BOOL
"M 18.3"	M 18.3	BOOL	// MARCA AUXILIAR - SIMULACION DE RETROAVISOS # 4
"M 18.4"	M 18.4	BOOL	// MARCA AUXILIAR - SIMULACION DE RETROAVISOS # 3
"M 18.5"	M 18.5	BOOL
"M 18.6"	M 18.6	BOOL
"M 18.7"	M 18.7	BOOL
"M 19.0"	M 19.0	BOOL
"M 19.1"	M 19.1	BOOL
"M 19.2"	M 19.2	BOOL
"M 19.3"	M 19.3	BOOL	// MARCA AUXILIAR - SIMULACION DE RETROAVISOS # 3
"M 19.4"	M 19.4	BOOL	// MARCA AUXILIAR - SIMULACION DE RETROAVISOS # 3
"M 19.5"	M 19.5	BOOL
"M 19.6"	M 19.6	BOOL
"M 19.7"	M 19.7	BOOL
"M 20.0"	M 20.0	BOOL
"M 20.1"	M 20.1	BOOL
"M 20.2"	M 20.2	BOOL
"M 20.3"	M 20.3	BOOL
"M 20.4"	M 20.4	BOOL
"M 20.5"	M 20.5	BOOL
"M 20.6"	M 20.6	BOOL
"M 20.7"	M 20.7	BOOL
"M 21.0"	M 21.0	BOOL
"M 21.1"	M 21.1	BOOL
"M 21.2"	M 21.2	BOOL
"M 21.3"	M 21.3	BOOL
"M 21.4"	M 21.4	BOOL
"M 21.5"	M 21.5	BOOL
"M 21.6"	M 21.6	BOOL
"M 21.7"	M 21.7	BOOL
"M 22.0"	M 22.0	BOOL
"M 22.1"	M 22.1	BOOL
"M 22.2"	M 22.2	BOOL
"M 22.3"	M 22.3	BOOL
"M 22.4"	M 22.4	BOOL
"M 22.5"	M 22.5	BOOL
"M 22.6"	M 22.6	BOOL
"M 22.7"	M 22.7	BOOL
"M 23.0"	M 23.0	BOOL
"M 23.1"	M 23.1	BOOL
"M 23.2"	M 23.2	BOOL
"M 23.3"	M 23.3	BOOL
"M 23.4"	M 23.4	BOOL
"M 23.5"	M 23.5	BOOL
"M 23.6"	M 23.6	BOOL
"M 23.7"	M 23.7	BOOL
"M 24.0"	M 24.0	BOOL
"M 24.1"	M 24.1	BOOL
"M 24.2"	M 24.2	BOOL
"M 24.3"	M 24.3	BOOL
"M 24.4"	M 24.4	BOOL
"M 24.5"	M 24.5	BOOL
"M 24.6"	M 24.6	BOOL
"M 24.7"	M 24.7	BOOL
"M 25.0"	M 25.0	BOOL
"M 25.1"	M 25.1	BOOL
"M 25.2"	M 25.2	BOOL
"M 25.3"	M 25.3	BOOL
"M 25.4"	M 25.4	BOOL
"M 25.5"	M 25.5	BOOL
"M 25.6"	M 25.6	BOOL
"M 25.7"	M 25.7	BOOL
"M 26.0"	M 26.0	BOOL
"M 26.1"	M 26.1	BOOL
"M 26.2"	M 26.2	BOOL
"M 26.3"	M 26.3	BOOL
"M 26.4"	M 26.4	BOOL
"M 26.5"	M 26.5	BOOL
"M 26.6"	M 26.6	BOOL
"M 26.7"	M 26.7	BOOL
"M 27.0"	M 27.0	BOOL
"M 27.1"	M 27.1	BOOL
"M 27.2"	M 27.2	BOOL
"M 27.3"	M 27.3	BOOL
"M 27.4"	M 27.4	BOOL
"M 27.5"	M 27.5	BOOL
"M 27.6"	M 27.6	BOOL
"M 27.7"	M 27.7	BOOL
"M 28.0"	M 28.0	BOOL
"M 28.1"	M 28.1	BOOL
"M 28.2"	M 28.2	BOOL
"M 28.3"	M 28.3	BOOL
"M 28.4"	M 28.4	BOOL
"M 28.5"	M 28.5	BOOL
"M 28.6"	M 28.6	BOOL
"M 28.7"	M 28.7	BOOL
"M 29.0"	M 29.0	BOOL
"M 29.1"	M 29.1	BOOL
"M 29.2"	M 29.2	BOOL
"M 29.3"	M 29.3	BOOL
"M 29.4"	M 29.4	BOOL
"M 29.5"	M 29.5	BOOL
"M 29.6"	M 29.6	BOOL
"M 29.7"	M 29.7	BOOL
"M 30.0"	M 30.0	BOOL
"M 30.1"	M 30.1	BOOL
"M 30.2"	M 30.2	BOOL
"M 30.3"	M 30.3	BOOL
"M 30.4"	M 30.4	BOOL
"M 30.5"	M 30.5	BOOL
"M 30.6"	M 30.6	BOOL
"M 30.7"	M 30.7	BOOL
"M 31.0"	M 31.0	BOOL
"M 31.1"	M 31.1	BOOL
"M 31.2"	M 31.2	BOOL
"M 31.3"	M 31.3	BOOL
"M 31.4"	M 31.4	BOOL
"M 31.5"	M 31.5	BOOL
"M 31.6"	M 31.6	BOOL
"M 31.7"	M 31.7	BOOL
"M 32.0"	M 32.0	BOOL
"M 32.1"	M 32.1	BOOL
"M 32.2"	M 32.2	BOOL
"M 32.3"	M 32.3	BOOL
"M 32.4"	M 32.4	BOOL
"M 32.5"	M 32.5	BOOL
"M 32.6"	M 32.6	BOOL
"M 32.7"	M 32.7	BOOL
"M 33.0"	M 33.0	BOOL
"M 33.1"	M 33.1	BOOL
"M 33.2"	M 33.2	BOOL
"M 33.3"	M 33.3	BOOL
"M 33.4"	M 33.4	BOOL
"M 33.5"	M 33.5	BOOL
"M 33.6"	M 33.6	BOOL
"M 33.7"	M 33.7	BOOL
"M 34.0"	M 34.0	BOOL
"M 34.1"	M 34.1	BOOL
"M 34.2"	M 34.2	BOOL
"M 34.3"	M 34.3	BOOL
"M 34.4"	M 34.4	BOOL
"M 34.5"	M 34.5	BOOL
"M 34.6"	M 34.6	BOOL
"M 34.7"	M 34.7	BOOL
"M 35.0"	M 35.0	BOOL
"M 35.1"	M 35.1	BOOL
"M 35.2"	M 35.2	BOOL
"M 35.3"	M 35.3	BOOL
"M 35.4"	M 35.4	BOOL
"M 35.5"	M 35.5	BOOL
"M 35.6"	M 35.6	BOOL
"M 35.7"	M 35.7	BOOL
"M 36.0"	M 36.0	BOOL
"M 36.1"	M 36.1	BOOL
"M 36.2"	M 36.2	BOOL
"M 36.3"	M 36.3	BOOL
"M 36.4"	M 36.4	BOOL
"M 36.5"	M 36.5	BOOL
"M 36.6"	M 36.6	BOOL
"M 36.7"	M 36.7	BOOL
"M 37.0"	M 37.0	BOOL
"M 37.1"	M 37.1	BOOL
"M 37.2"	M 37.2	BOOL
"M 37.3"	M 37.3	BOOL
"M 37.4"	M 37.4	BOOL
"M 37.5"	M 37.5	BOOL
"M 37.6"	M 37.6	BOOL
"M 37.7"	M 37.7	BOOL
"M 38.0"	M 38.0	BOOL
"M 38.1"	M 38.1	BOOL
"M 38.2"	M 38.2	BOOL
"M 38.3"	M 38.3	BOOL
"M 38.4"	M 38.4	BOOL
"M 38.5"	M 38.5	BOOL
"M 38.6"	M 38.6	BOOL
"M 38.7"	M 38.7	BOOL
"M 39.0"	M 39.0	BOOL
"M 39.1"	M 39.1	BOOL
"M 39.2"	M 39.2	BOOL
"M 39.3"	M 39.3	BOOL
"M 39.4"	M 39.4	BOOL
"M 39.5"	M 39.5	BOOL
"M 39.6"	M 39.6	BOOL
"M 39.7"	M 39.7	BOOL
"M 40.0"	M 40.0	BOOL	// OSCILADOR DE SEMAFORO - PARTE 1
"M 40.1"	M 40.1	BOOL	// OSCILADOR DE SEMAFORO - PARTE 2
"M 41.0"	M 41.0	BOOL
"M 41.1"	M 41.1	BOOL
"M 41.2"	M 41.2	BOOL
"M 41.3"	M 41.3	BOOL
"M 41.4"	M 41.4	BOOL
"M 41.6"	M 41.6	BOOL	// INDICACION DE SEMAFORO - LUZ VERDE - PARTE 1
"M 41.7"	M 41.7	BOOL	// INDICACION DE SEMAFORO - FLECHA LUZ VERDE - PARTE 1
"M 42.0"	M 42.0	BOOL	// SEMAFORO # 4 INDICACIONES - LUZ ROJA ( MARCA AUXILIAR )
"M 42.1"	M 42.1	BOOL	// SEMAFORO # 4 INDICACIONES - LUZ VERDE ( MARCA AUXILIAR )
"M 42.2"	M 42.2	BOOL	// SEMAFORO # 4 INDICACIONES - LUZ AMARILLA ( MARCA AUXILIAR )
"M 42.3"	M 42.3	BOOL	// SEMAFORO # 4 INDICACIONES - FLECHA_LUZ VERDE ( MARCA AUXILIAR )
"M 43.0"	M 43.0	BOOL	// TEMPORIZADOR EN OPERACION ( INICIO DE SECUENCIA )
"M 43.1"	M 43.1	BOOL	// TEMPORIZADOR EN OPERACION ( INDICACION DE LUZ ROJA )
"M 43.2"	M 43.2	BOOL
"M 43.3"	M 43.3	BOOL
"M 43.4"	M 43.4	BOOL	// TEMPORIZADOR EN OPERACION ( INDICACION DE FLECHA )
"M 44.0"	M 44.0	BOOL	// SEMAFORO # 3 INDICACIONES - LUZ ROJA ( MARCA AUXILIAR )
"M 44.1"	M 44.1	BOOL	// SEMAFORO # 3 INDICACIONES - LUZ VERDE ( MARCA AUXILIAR )
"M 44.2"	M 44.2	BOOL	// SEMAFORO # 3 INDICACIONES - LUZ AMARILLA ( MARCA AUXILIAR )
"M 44.6"	M 44.6	BOOL
"M 46.0"	M 46.0	BOOL	// FIN DE TIEMPO DE DURACION ( LUZ ROJA )
"M 46.1"	M 46.1	BOOL	// FIN DE TIEMPO DE DURACION ( LUZ VERDE )
"M 46.2"	M 46.2	BOOL	// FIN DE TIEMPO DE DURACION ( LUZ AMARILLA )
"M 46.3"	M 46.3	BOOL	// TEMPORIZADOR DE LUZ VERDE - FUNCIONANDO
"M 50.0"	M 50.0	BOOL	// FRECUENCIA DE 2 HZ
"M 50.1"	M 50.1	BOOL	// FRECUENCIA DE 1 HZ
"M 50.2"	M 50.2	BOOL	// FRECUENCIA DE 0.5 HZ
"M 50.3"	M 50.3	BOOL	// FRECUENCIA DE 0.5 HZ
"M 51.0"	M 51.0	BOOL	// CONDICION No. 1 - AL MENOS DOS O TRES VENTILADORES FUNCIONAN
"M 51.1"	M 51.1	BOOL	// CONDICION No. 2 - NO FUNCIONA NINGUN VENTILADOR
"M 51.2"	M 51.2	BOOL	// CONDICION No. 3 - SOLAMENTE FUNCIONA UN VENTILADOR
"M 51.3"	M 51.3	BOOL
"M 51.4"	M 51.4	BOOL	// SISTEMA EN OPERACION
"M 51.5"	M 51.5	BOOL	// INDICACION DE LAMPARA DE SUPERVISION
"M 52.0"	M 52.0	BOOL	// DESCONEXION DE LA SUPERVISION
"M 52.1"	M 52.1	BOOL	// TIEMPO DE SUPERVISION DE FRECUENCIA - ACTIVADO
"M 52.2"	M 52.2	BOOL	// INDICACION DE FALLA DE SUPERVISION
"M 52.3"	M 52.3	BOOL	// ACUSE DE AVISO
"M 53.0"	M 53.0	BOOL	// MARCA AUXILIAR DEL FLANCO POSITIVO
"M 53.1"	M 53.1	BOOL	// MARCA AUXILIAR DEL FLANCO NEGATIVO
"M 53.2"	M 53.2	BOOL	// ARMARIO DE ILUMINACION B
"M 53.3"	M 53.3	BOOL	// ARMARIO DE ILUMINACION A
"M 53.4"	M 53.4	BOOL	// INDICACION DE RECINTO OCUPADO
"M 53.5"	M 53.5	BOOL	// VALOR DE AJUSTE DEL CONTADOR ( IMPULSO )
"M 53.6"	M 53.6	BOOL	// FLANCO NEGATIVO ( - )
"M 53.7"	M 53.7	BOOL	// FLANCO POSITIVO ( + )
"M 59.0"	M 59.0	BOOL	// CONTADOR = 1
"M 59.1"	M 59.1	BOOL	// CONTADOR = 2
"M 59.2"	M 59.2	BOOL	// CONTADOR = 4
"M 59.3"	M 59.3	BOOL	// CONTADOR = 8 SE CONMUTA AL ESTADO DE CONTADOR = 0
"M 60.0"	M 60.0	BOOL	// GENERADOR DE IMPULSOS ( PARTE I )
"M 60.1"	M 60.1	BOOL	// GENERADOR DE IMPULSOS ( PARTE II )
"M 60.2"	M 60.2	BOOL	// SEMAFORO - TIEMPO DE INDICACION ( LUZ ROJA )
"M 60.3"	M 60.3	BOOL	// SEMAFORO - TIEMPO DE INDICACION ( LUZ VERDE )
"M 60.4"	M 60.4	BOOL	// SEMAFORO - TIEMPO DE INDICACION ( LUZ AMARILLA )
"M 61.0"	M 61.0	BOOL	// MARCA AUXILIAR - INDICACION LUZ ROJA
"M 61.1"	M 61.1	BOOL	// MARCA AUXILIAR - INDICACION LUZ VERDE - PARTE I
"M 61.2"	M 61.2	BOOL	// MARCA AUXILIAR - INDICACION LUZ VERDE - PARTE II
"M 61.3"	M 61.3	BOOL	// MARCA AUXILIAR - INDICACION LUZ AMARILLA
"M 80.0"	M 80.0	BOOL
"M 80.1"	M 80.1	BOOL	// MARCA AUXILAIR - FLANCO POSITIVO
"M 80.2"	M 80.2	BOOL	// MARCA AUXILIAR - FLANCO NEGATIVO
"M 80.3"	M 80.3	BOOL	// FLANCO POSITIVO
"M 80.4"	M 80.4	BOOL	// FLANCO NEGATIVO
"M 80.5"	M 80.5	BOOL	// MARCA AUXILIAR - AVANZAR
"M 80.6"	M 80.6	BOOL	// MARCA AUXILIAR  - REGRESAR
"M 99.1"	M 99.1	BOOL	// MARCA AUXILIAR DE FLANCO POSITIVO
"M 99.2"	M 99.2	BOOL	// MARCA FLANCO POSITIVO ( + )
"M 99.3"	M 99.3	BOOL	// MARCA AUXILIAR DE FLANCO NEGATIVO
"M 99.4"	M 99.4	BOOL	// MARCA DE FLANCO NEGATIVO ( - )
"M 99.5"	M 99.5	BOOL	// MARCA DE EVALUACION DEFLANCOS
"M 101.0"	M 101.0	BOOL	// MARCA AUXILIAR - SELECTOR EN POSICION FUERA
"M 101.1"	M 101.1	BOOL	// MARCA AUXILIAR - SELECTOR EN MODO LOCAL
"M 101.2"	M 101.2	BOOL	// MARCA AUXILIAR - SELECTOR EN MODO REMOTO
"M 102.0"	M 102.0	BOOL	// MARCA AUXILIAR - SELECTOR EN POSICION FUERA
"M 102.1"	M 102.1	BOOL	// MARCA AUXILIAR - SELECTOR EN MODO LOCAL
"M 102.2"	M 102.2	BOOL	// MARCA AUXILIAR - SELECTOR EN MODO REMOTO
"M 103.0"	M 103.0	BOOL	// MARCA AUXILIAR - SELECTOR EN POSICION FUERA
"M 103.1"	M 103.1	BOOL	// MARCA AUXILIAR - SELECTOR EN MODO LOCAL
"M 103.2"	M 103.2	BOOL	// MARCA AUXILIAR - SELECTOR EN MODO REMOTO
"M 104.0"	M 104.0	BOOL	// MARCA AUXILIAR - SELECTOR EN POSICION FUERA
"M 104.1"	M 104.1	BOOL	// MARCA AUXILIAR - SELECTOR EN MODO LOCAL
"M 104.2"	M 104.2	BOOL	// MARCA AUXILIAR - SELECTOR EN MODO REMOTO
"M 105.0"	M 105.0	BOOL	// MARCA AUXILIAR - SELECTOR EN POSICION FUERA
"M 105.1"	M 105.1	BOOL	// MARCA AUXILIAR - SELECTOR EN MODO LOCAL
"M 105.2"	M 105.2	BOOL	// MARCA AUXILIAR - SELECTOR EN MODO REMOTO
"M 106.0"	M 106.0	BOOL	// MARCA AUXILIAR - SELECTOR EN POSICION FUERA
"M 106.1"	M 106.1	BOOL	// MARCA AUXILIAR - SELECTOR EN MODO LOCAL
"M 106.2"	M 106.2	BOOL	// MARCA AUXILIAR - SELECTOR EN MODO REMOTO
"M 107.0"	M 107.0	BOOL	// MARCA AUXILIAR - SELECTOR EN POSICION FUERA
"M 107.1"	M 107.1	BOOL	// MARCA AUXILIAR - SELECTOR EN MODO LOCAL
"M 107.2"	M 107.2	BOOL	// MARCA AUXILIAR - SELECTOR EN MODO REMOTO
"M 108.0"	M 108.0	BOOL	// MARCA AUXILIAR - SELECTOR EN POSICION FUERA
"M 108.1"	M 108.1	BOOL	// MARCA AUXILIAR - SELECTOR EN MODO LOCAL
"M 108.2"	M 108.2	BOOL	// MARCA AUXILIAR - SELECTOR EN MODO REMOTO
"M 111.0"	M 111.0	BOOL	// MARCA AUXILIAR - CONTACTOR DESCONECTADO
"M 111.1"	M 111.1	BOOL	// MARCA AUXILIAR - CONTACTOR CONECTADO
"M 112.0"	M 112.0	BOOL	// MARCA AUXILIAR - CONTACTOR DESCONECTADO
"M 112.1"	M 112.1	BOOL	// MARCA AUXILIAR - CONTACTOR CONECTADO
"M 113.0"	M 113.0	BOOL	// MARCA AUXILIAR - CONTACTOR DESCONECTADO
"M 113.1"	M 113.1	BOOL	// MARCA AUXILIAR - CONTACTOR CONECTADO
"M 114.0"	M 114.0	BOOL	// MARCA AUXILIAR - CONTACTOR DESCONECTADO
"M 114.1"	M 114.1	BOOL	// MARCA AUXILIAR - CONTACTOR CONECTADO
"M 115.0"	M 115.0	BOOL	// MARCA AUXILIAR - CONTACTOR DESCONECTADO
"M 115.1"	M 115.1	BOOL	// MARCA AUXILIAR - CONTACTOR CONECTADO
"M 116.0"	M 116.0	BOOL	// MARCA AUXILIAR - CONTACTOR DESCONECTADO
"M 116.1"	M 116.1	BOOL	// MARCA AUXILIAR - CONTACTOR CONECTADO
"M 117.0"	M 117.0	BOOL	// MARCA AUXILIAR - CONTACTOR DESCONECTADO
"M 117.1"	M 117.1	BOOL	// MARCA AUXILIAR - CONTACTOR CONECTADO
"M 118.0"	M 118.0	BOOL	// MARCA AUXILIAR - CONTACTOR DESCONECTADO
"M 118.1"	M 118.1	BOOL	// MARCA AUXILIAR - CONTACTOR CONECTADO
"M 119.0"	M 119.0	BOOL	// MARCA AUXILIAR - CONTACTOR DESCONECTADO
"M 119.1"	M 119.1	BOOL	// MARCA AUXILIAR - CONTACTOR CONECTADO
"M 120.0"	M 120.0	BOOL
"M 120.1"	M 120.1	BOOL
"M 120.2"	M 120.2	BOOL
"M 120.3"	M 120.3	BOOL
"M 120.4"	M 120.4	BOOL
"M 120.5"	M 120.5	BOOL
"M 120.6"	M 120.6	BOOL
"M 120.7"	M 120.7	BOOL
"M 121.0"	M 121.0	BOOL
"M 121.1"	M 121.1	BOOL
"M 121.2"	M 121.2	BOOL
"M 121.3"	M 121.3	BOOL
"M 121.4"	M 121.4	BOOL
"M 121.5"	M 121.5	BOOL
"M 121.6"	M 121.6	BOOL
"M 121.7"	M 121.7	BOOL
"M 122.0"	M 122.0	BOOL
"M 122.1"	M 122.1	BOOL
"M 122.2"	M 122.2	BOOL
"M 122.3"	M 122.3	BOOL
"M 122.4"	M 122.4	BOOL
"M 122.5"	M 122.5	BOOL
"M 122.6"	M 122.6	BOOL
"M 122.7"	M 122.7	BOOL
"M 123.0"	M 123.0	BOOL
"M 123.1"	M 123.1	BOOL
"M 123.2"	M 123.2	BOOL
"M 123.3"	M 123.3	BOOL
"M 123.4"	M 123.4	BOOL
"M 123.5"	M 123.5	BOOL
"M 123.6"	M 123.6	BOOL
"M 123.7"	M 123.7	BOOL
"M 124.0"	M 124.0	BOOL
"M 124.1"	M 124.1	BOOL
"M 124.2"	M 124.2	BOOL
"M 124.3"	M 124.3	BOOL
"M 124.4"	M 124.4	BOOL
"M 124.5"	M 124.5	BOOL
"M 124.6"	M 124.6	BOOL
"M 124.7"	M 124.7	BOOL
"M 125.0"	M 125.0	BOOL
"M 125.1"	M 125.1	BOOL
"M 125.2"	M 125.2	BOOL
"M 125.3"	M 125.3	BOOL
"M 125.4"	M 125.4	BOOL
"M 125.5"	M 125.5	BOOL
"M 125.6"	M 125.6	BOOL
"M 125.7"	M 125.7	BOOL
"M 126.0"	M 126.0	BOOL
"M 126.1"	M 126.1	BOOL
"M 126.2"	M 126.2	BOOL
"M 126.3"	M 126.3	BOOL
"M 126.4"	M 126.4	BOOL
"M 126.5"	M 126.5	BOOL
"M 126.6"	M 126.6	BOOL
"M 126.7"	M 126.7	BOOL
"M 127.0"	M 127.0	BOOL
"M 127.1"	M 127.1	BOOL
"M 127.2"	M 127.2	BOOL
"M 127.3"	M 127.3	BOOL
"M 127.4"	M 127.4	BOOL
"M 127.5"	M 127.5	BOOL
"M 127.6"	M 127.6	BOOL
"M 127.7"	M 127.7	BOOL
"M 128.0"	M 128.0	BOOL
"M 128.1"	M 128.1	BOOL
"M 128.2"	M 128.2	BOOL
"M 128.3"	M 128.3	BOOL
"M 128.4"	M 128.4	BOOL
"M 128.5"	M 128.5	BOOL
"M 128.6"	M 128.6	BOOL
"M 128.7"	M 128.7	BOOL
"M 129.0"	M 129.0	BOOL
"M 129.1"	M 129.1	BOOL
"M 129.2"	M 129.2	BOOL
"M 129.3"	M 129.3	BOOL
"M 129.4"	M 129.4	BOOL
"M 129.5"	M 129.5	BOOL
"M 129.6"	M 129.6	BOOL
"M 129.7"	M 129.7	BOOL
"M 130.0"	M 130.0	BOOL
"M 130.1"	M 130.1	BOOL
"M 130.2"	M 130.2	BOOL
"M 130.3"	M 130.3	BOOL
"M 130.4"	M 130.4	BOOL
"M 130.5"	M 130.5	BOOL
"M 130.6"	M 130.6	BOOL
"M 130.7"	M 130.7	BOOL
"M 131.0"	M 131.0	BOOL
"M 131.1"	M 131.1	BOOL
"M 131.2"	M 131.2	BOOL
"M 131.3"	M 131.3	BOOL
"M 131.4"	M 131.4	BOOL
"M 131.5"	M 131.5	BOOL
"M 131.6"	M 131.6	BOOL
"M 131.7"	M 131.7	BOOL
"M 132.0"	M 132.0	BOOL
"M 132.1"	M 132.1	BOOL
"M 132.2"	M 132.2	BOOL
"M 132.3"	M 132.3	BOOL
"M 132.4"	M 132.4	BOOL
"M 132.5"	M 132.5	BOOL
"M 132.6"	M 132.6	BOOL
"M 132.7"	M 132.7	BOOL
"M 133.0"	M 133.0	BOOL
"M 133.1"	M 133.1	BOOL
"M 133.2"	M 133.2	BOOL
"M 133.3"	M 133.3	BOOL
"M 133.4"	M 133.4	BOOL
"M 133.5"	M 133.5	BOOL
"M 133.6"	M 133.6	BOOL
"M 133.7"	M 133.7	BOOL
"M 134.0"	M 134.0	BOOL
"M 134.1"	M 134.1	BOOL
"M 134.2"	M 134.2	BOOL
"M 134.3"	M 134.3	BOOL
"M 134.4"	M 134.4	BOOL
"M 134.5"	M 134.5	BOOL
"M 134.6"	M 134.6	BOOL
"M 134.7"	M 134.7	BOOL
"M 135.0"	M 135.0	BOOL
"M 135.1"	M 135.1	BOOL
"M 135.2"	M 135.2	BOOL
"M 135.3"	M 135.3	BOOL
"M 135.4"	M 135.4	BOOL
"M 135.5"	M 135.5	BOOL
"M 135.6"	M 135.6	BOOL
"M 135.7"	M 135.7	BOOL
"M 136.0"	M 136.0	BOOL
"M 136.1"	M 136.1	BOOL
"M 136.2"	M 136.2	BOOL
"M 136.3"	M 136.3	BOOL
"M 136.4"	M 136.4	BOOL
"M 136.5"	M 136.5	BOOL
"M 136.6"	M 136.6	BOOL
"M 136.7"	M 136.7	BOOL
"M 137.0"	M 137.0	BOOL
"M 137.1"	M 137.1	BOOL
"M 137.2"	M 137.2	BOOL
"M 137.3"	M 137.3	BOOL
"M 137.4"	M 137.4	BOOL
"M 137.5"	M 137.5	BOOL
"M 137.6"	M 137.6	BOOL
"M 137.7"	M 137.7	BOOL
"M 138.0"	M 138.0	BOOL	// ENCENDER BOCINA - ALARMA ACTIVADA
"M 138.1"	M 138.1	BOOL	// MARCA AUXILIAR - PUNTO DE AJUSTE
"M 138.2"	M 138.2	BOOL	// FLANCO POSITIVO ( + ) - PUNTO DE AJUSTE
"M 138.3"	M 138.3	BOOL	// REINICIO DE BOCINA
"M 138.4"	M 138.4	BOOL	// MARCA AUXILIAR - BOCINA ACTIVADA
"M 138.5"	M 138.5	BOOL
"M 138.6"	M 138.6	BOOL
"M 138.7"	M 138.7	BOOL
"M 139.0"	M 139.0	BOOL	// BOTON DE AJUSTE DE ALARMA
"M 139.1"	M 139.1	BOOL	// BOTON DE SUBIR MINUTOS
"M 139.2"	M 139.2	BOOL	// BOTON DE SUBIR HORAS
"M 139.3"	M 139.3	BOOL	// BOTON DE AJUSTE DE RELOJ
"M 139.4"	M 139.4	BOOL	// BOTON SELECTOR DE ALARMA ACTIVADA
"M 139.5"	M 139.5	BOOL	// BOTON DE SILENCIAR BOCINA
"M 139.6"	M 139.6	BOOL
"M 139.7"	M 139.7	BOOL	// INDICACION DE BOCINA
"M 140.0"	M 140.0	BOOL
"M 140.1"	M 140.1	BOOL
"M 140.2"	M 140.2	BOOL
"M 140.3"	M 140.3	BOOL
"M 140.4"	M 140.4	BOOL
"M 140.5"	M 140.5	BOOL
"M 140.6"	M 140.6	BOOL
"M 140.7"	M 140.7	BOOL
"M 141.0"	M 141.0	BOOL
"M 141.1"	M 141.1	BOOL
"M 141.2"	M 141.2	BOOL
"M 141.3"	M 141.3	BOOL
"M 141.4"	M 141.4	BOOL
"M 141.5"	M 141.5	BOOL
"M 141.6"	M 141.6	BOOL
"M 141.7"	M 141.7	BOOL
"M 142.0"	M 142.0	BOOL
"M 142.1"	M 142.1	BOOL
"M 142.2"	M 142.2	BOOL
"M 142.3"	M 142.3	BOOL
"M 142.4"	M 142.4	BOOL
"M 142.5"	M 142.5	BOOL
"M 142.6"	M 142.6	BOOL
"M 142.7"	M 142.7	BOOL
"M 143.0"	M 143.0	BOOL
"M 143.1"	M 143.1	BOOL
"M 143.2"	M 143.2	BOOL
"M 143.3"	M 143.3	BOOL
"M 143.4"	M 143.4	BOOL
"M 143.5"	M 143.5	BOOL
"M 143.6"	M 143.6	BOOL
"M 143.7"	M 143.7	BOOL
"M 144.0"	M 144.0	BOOL	// ENCENDER BOCINA - ALARMA ACTIVADA
"M 144.1"	M 144.1	BOOL	// MARCA AUXILIAR - PUNTO DE AJUSTE
"M 144.2"	M 144.2	BOOL	// FLANCO POSITIVO ( + ) - PUNTO DE AJUSTE
"M 144.3"	M 144.3	BOOL	// REINICIO DE BOCINA
"M 144.4"	M 144.4	BOOL	// MARCA AUXILIAR - BOCINA ACTIVADA
"M 144.5"	M 144.5	BOOL
"M 144.6"	M 144.6	BOOL
"M 144.7"	M 144.7	BOOL
"M 145.0"	M 145.0	BOOL
"M 145.1"	M 145.1	BOOL
"M 145.2"	M 145.2	BOOL
"M 145.3"	M 145.3	BOOL
"M 145.4"	M 145.4	BOOL
"M 145.5"	M 145.5	BOOL
"M 145.6"	M 145.6	BOOL
"M 145.7"	M 145.7	BOOL
"M 146.0"	M 146.0	BOOL
"M 146.1"	M 146.1	BOOL
"M 146.2"	M 146.2	BOOL
"M 146.3"	M 146.3	BOOL
"M 146.4"	M 146.4	BOOL
"M 146.5"	M 146.5	BOOL
"M 146.6"	M 146.6	BOOL
"M 146.7"	M 146.7	BOOL
"M 147.0"	M 147.0	BOOL
"M 147.1"	M 147.1	BOOL
"M 147.2"	M 147.2	BOOL
"M 147.3"	M 147.3	BOOL
"M 147.4"	M 147.4	BOOL
"M 147.5"	M 147.5	BOOL
"M 147.6"	M 147.6	BOOL
"M 147.7"	M 147.7	BOOL
"M 148.0"	M 148.0	BOOL
"M 148.1"	M 148.1	BOOL
"M 148.2"	M 148.2	BOOL
"M 148.3"	M 148.3	BOOL
"M 148.4"	M 148.4	BOOL
"M 148.5"	M 148.5	BOOL
"M 148.6"	M 148.6	BOOL
"M 148.7"	M 148.7	BOOL
"M 149.0"	M 149.0	BOOL
"M 149.1"	M 149.1	BOOL
"M 149.2"	M 149.2	BOOL
"M 149.3"	M 149.3	BOOL
"M 149.4"	M 149.4	BOOL
"M 149.5"	M 149.5	BOOL
"M 149.6"	M 149.6	BOOL
"M 149.7"	M 149.7	BOOL
"M 150.0"	M 150.0	BOOL
"M 150.1"	M 150.1	BOOL
"M 150.2"	M 150.2	BOOL
"M 150.3"	M 150.3	BOOL
"M 150.4"	M 150.4	BOOL
"M 150.5"	M 150.5	BOOL
"M 150.6"	M 150.6	BOOL
"M 150.7"	M 150.7	BOOL
"M 151.0"	M 151.0	BOOL
"M 151.1"	M 151.1	BOOL
"M 151.2"	M 151.2	BOOL
"M 151.3"	M 151.3	BOOL
"M 151.4"	M 151.4	BOOL
"M 151.5"	M 151.5	BOOL
"M 151.6"	M 151.6	BOOL
"M 151.7"	M 151.7	BOOL
"M 152.0"	M 152.0	BOOL
"M 152.1"	M 152.1	BOOL
"M 152.2"	M 152.2	BOOL
"M 152.3"	M 152.3	BOOL
"M 152.4"	M 152.4	BOOL
"M 152.5"	M 152.5	BOOL
"M 152.6"	M 152.6	BOOL
"M 152.7"	M 152.7	BOOL
"M 153.0"	M 153.0	BOOL
"M 153.1"	M 153.1	BOOL
"M 153.2"	M 153.2	BOOL
"M 153.3"	M 153.3	BOOL
"M 153.4"	M 153.4	BOOL
"M 153.5"	M 153.5	BOOL
"M 153.6"	M 153.6	BOOL
"M 153.7"	M 153.7	BOOL
"M 154.0"	M 154.0	BOOL
"M 154.1"	M 154.1	BOOL
"M 154.2"	M 154.2	BOOL
"M 154.3"	M 154.3	BOOL
"M 154.4"	M 154.4	BOOL
"M 154.5"	M 154.5	BOOL
"M 154.6"	M 154.6	BOOL
"M 154.7"	M 154.7	BOOL
"M 155.0"	M 155.0	BOOL
"M 155.1"	M 155.1	BOOL
"M 155.2"	M 155.2	BOOL
"M 155.3"	M 155.3	BOOL
"M 155.4"	M 155.4	BOOL
"M 155.5"	M 155.5	BOOL
"M 155.6"	M 155.6	BOOL
"M 155.7"	M 155.7	BOOL
"M 156.0"	M 156.0	BOOL
"M 156.1"	M 156.1	BOOL
"M 156.2"	M 156.2	BOOL
"M 156.3"	M 156.3	BOOL
"M 156.4"	M 156.4	BOOL
"M 156.5"	M 156.5	BOOL
"M 156.6"	M 156.6	BOOL
"M 156.7"	M 156.7	BOOL
"M 157.0"	M 157.0	BOOL
"M 157.1"	M 157.1	BOOL
"M 157.2"	M 157.2	BOOL
"M 157.3"	M 157.3	BOOL
"M 157.4"	M 157.4	BOOL
"M 157.5"	M 157.5	BOOL
"M 157.6"	M 157.6	BOOL
"M 157.7"	M 157.7	BOOL
"M 158.0"	M 158.0	BOOL
"M 158.1"	M 158.1	BOOL
"M 158.2"	M 158.2	BOOL
"M 158.3"	M 158.3	BOOL
"M 158.4"	M 158.4	BOOL
"M 158.5"	M 158.5	BOOL
"M 158.6"	M 158.6	BOOL
"M 158.7"	M 158.7	BOOL
"M 159.0"	M 159.0	BOOL
"M 159.1"	M 159.1	BOOL
"M 159.2"	M 159.2	BOOL
"M 159.3"	M 159.3	BOOL
"M 159.4"	M 159.4	BOOL
"M 159.5"	M 159.5	BOOL
"M 159.6"	M 159.6	BOOL
"M 159.7"	M 159.7	BOOL
"M 160.0"	M 160.0	BOOL
"M 160.1"	M 160.1	BOOL
"M 160.2"	M 160.2	BOOL
"M 160.3"	M 160.3	BOOL
"M 160.4"	M 160.4	BOOL
"M 160.5"	M 160.5	BOOL
"M 160.6"	M 160.6	BOOL
"M 160.7"	M 160.7	BOOL
"M 161.0"	M 161.0	BOOL
"M 161.1"	M 161.1	BOOL
"M 161.2"	M 161.2	BOOL
"M 161.3"	M 161.3	BOOL
"M 161.4"	M 161.4	BOOL
"M 161.5"	M 161.5	BOOL
"M 161.6"	M 161.6	BOOL
"M 161.7"	M 161.7	BOOL
"M 162.0"	M 162.0	BOOL
"M 162.1"	M 162.1	BOOL
"M 162.2"	M 162.2	BOOL
"M 162.3"	M 162.3	BOOL
"M 162.4"	M 162.4	BOOL
"M 162.5"	M 162.5	BOOL
"M 162.6"	M 162.6	BOOL
"M 162.7"	M 162.7	BOOL
"M 163.0"	M 163.0	BOOL
"M 163.1"	M 163.1	BOOL
"M 163.2"	M 163.2	BOOL
"M 163.3"	M 163.3	BOOL
"M 163.4"	M 163.4	BOOL
"M 163.5"	M 163.5	BOOL
"M 163.6"	M 163.6	BOOL
"M 163.7"	M 163.7	BOOL
"M 164.0"	M 164.0	BOOL
"M 164.1"	M 164.1	BOOL
"M 164.2"	M 164.2	BOOL
"M 164.3"	M 164.3	BOOL
"M 164.4"	M 164.4	BOOL
"M 164.5"	M 164.5	BOOL
"M 164.6"	M 164.6	BOOL
"M 164.7"	M 164.7	BOOL
"M 165.0"	M 165.0	BOOL
"M 165.1"	M 165.1	BOOL
"M 165.2"	M 165.2	BOOL
"M 165.3"	M 165.3	BOOL
"M 165.4"	M 165.4	BOOL
"M 165.5"	M 165.5	BOOL
"M 165.6"	M 165.6	BOOL
"M 165.7"	M 165.7	BOOL
"M 166.0"	M 166.0	BOOL
"M 166.1"	M 166.1	BOOL
"M 166.2"	M 166.2	BOOL
"M 166.3"	M 166.3	BOOL
"M 166.4"	M 166.4	BOOL
"M 166.5"	M 166.5	BOOL
"M 166.6"	M 166.6	BOOL
"M 166.7"	M 166.7	BOOL
"M 167.0"	M 167.0	BOOL
"M 167.1"	M 167.1	BOOL
"M 167.2"	M 167.2	BOOL
"M 167.3"	M 167.3	BOOL
"M 167.4"	M 167.4	BOOL
"M 167.5"	M 167.5	BOOL
"M 167.6"	M 167.6	BOOL
"M 167.7"	M 167.7	BOOL
"M 168.0"	M 168.0	BOOL
"M 168.1"	M 168.1	BOOL
"M 168.2"	M 168.2	BOOL
"M 168.3"	M 168.3	BOOL
"M 168.4"	M 168.4	BOOL
"M 168.5"	M 168.5	BOOL
"M 168.6"	M 168.6	BOOL
"M 168.7"	M 168.7	BOOL
"M 169.0"	M 169.0	BOOL
"M 169.1"	M 169.1	BOOL
"M 169.2"	M 169.2	BOOL
"M 169.3"	M 169.3	BOOL
"M 169.4"	M 169.4	BOOL
"M 169.5"	M 169.5	BOOL
"M 169.6"	M 169.6	BOOL
"M 169.7"	M 169.7	BOOL
"M 170.0"	M 170.0	BOOL	// ALARMA No. 1
"M 170.1"	M 170.1	BOOL	// ALARMA No. 2
"M 170.2"	M 170.2	BOOL	// ALARMA No. 3
"M 170.3"	M 170.3	BOOL	// ALARMA No. 4
"M 170.4"	M 170.4	BOOL	// ALARMA No. 5
"M 170.5"	M 170.5	BOOL	// ALARMA No. 6
"M 170.6"	M 170.6	BOOL	// ALARMA No. 7
"M 170.7"	M 170.7	BOOL	// ALARMA No. 8
"M 171.0"	M 171.0	BOOL	// FLANCO NEGATIVO ( - ) - ALARMA No. 1
"M 171.1"	M 171.1	BOOL	// MARCA AUXILIAR - ALARMA No. 1
"M 171.2"	M 171.2	BOOL	// MARCA AUXILIAR - RECONOCIMIENTO DE ALARMA No. 1
"M 171.3"	M 171.3	BOOL	// MARCA AUXILIAR - RESTABLECIMIENTO DE ALARMA No. 1
"M 171.4"	M 171.4	BOOL	// MARCA AUXILIAR - INDICACION DE ALARMA No. 1
"M 171.5"	M 171.5	BOOL
"M 171.6"	M 171.6	BOOL
"M 171.7"	M 171.7	BOOL
"M 172.0"	M 172.0	BOOL	// FLANCO NEGATIVO ( - ) - ALARMA No. 2
"M 172.1"	M 172.1	BOOL	// MARCA AUXILIAR - ALARMA No. 2
"M 172.2"	M 172.2	BOOL	// MARCA AUXILIAR - RECONOCIMIENTO DE ALARMA No. 2
"M 172.3"	M 172.3	BOOL	// MARCA AUXILIAR - RESTABLECIMIENTO DE ALARMA No. 2
"M 172.4"	M 172.4	BOOL	// MARCA AUXILIAR - INDICACION DE ALARMA No. 2
"M 172.5"	M 172.5	BOOL
"M 172.6"	M 172.6	BOOL
"M 172.7"	M 172.7	BOOL
"M 173.0"	M 173.0	BOOL	// FLANCO NEGATIVO ( - ) - ALARMA No. 3
"M 173.1"	M 173.1	BOOL	// MARCA AUXILIAR - ALARMA No. 3
"M 173.2"	M 173.2	BOOL	// MARCA AUXILIAR - RECONOCIMIENTO DE ALARMA No. 3
"M 173.3"	M 173.3	BOOL	// MARCA AUXILIAR - RESTABLECIMIENTO DE ALARMA No. 3
"M 173.4"	M 173.4	BOOL	// MARCA AUXILIAR - INDICACION DE ALARMA No. 3
"M 173.5"	M 173.5	BOOL
"M 173.6"	M 173.6	BOOL
"M 173.7"	M 173.7	BOOL
"M 174.0"	M 174.0	BOOL	// FLANCO NEGATIVO ( - ) - ALARMA No. 4
"M 174.1"	M 174.1	BOOL	// MARCA AUXILIAR - ALARMA No. 4
"M 174.2"	M 174.2	BOOL	// MARCA AUXILIAR - RECONOCIMIENTO DE ALARMA No. 4
"M 174.3"	M 174.3	BOOL	// MARCA AUXILIAR - RESTABLECIMIENTO DE ALARMA No. 4
"M 174.4"	M 174.4	BOOL	// MARCA AUXILIAR - INDICACION DE ALARMA No. 4
"M 174.5"	M 174.5	BOOL
"M 174.6"	M 174.6	BOOL
"M 174.7"	M 174.7	BOOL
"M 175.0"	M 175.0	BOOL	// FLANCO NEGATIVO ( - ) - ALARMA No. 5
"M 175.1"	M 175.1	BOOL	// MARCA AUXILIAR - ALARMA No. 5
"M 175.2"	M 175.2	BOOL	// MARCA AUXILIAR - RECONOCIMIENTO DE ALARMA No. 5
"M 175.3"	M 175.3	BOOL	// MARCA AUXILIAR - RESTABLECIMIENTO DE ALARMA No. 5
"M 175.4"	M 175.4	BOOL	// MARCA AUXILIAR - INDICACION DE ALARMA No. 5
"M 175.5"	M 175.5	BOOL
"M 175.6"	M 175.6	BOOL
"M 175.7"	M 175.7	BOOL
"M 176.0"	M 176.0	BOOL	// FLANCO NEGATIVO ( - ) - ALARMA No. 6
"M 176.1"	M 176.1	BOOL	// MARCA AUXILIAR - ALARMA No. 6
"M 176.2"	M 176.2	BOOL	// MARCA AUXILIAR - RECONOCIMIENTO DE ALARMA No. 6
"M 176.3"	M 176.3	BOOL	// MARCA AUXILIAR - RESTABLECIMIENTO DE ALARMA No. 6
"M 176.4"	M 176.4	BOOL	// MARCA AUXILIAR - INDICACION DE ALARMA No. 6
"M 176.5"	M 176.5	BOOL
"M 176.6"	M 176.6	BOOL
"M 176.7"	M 176.7	BOOL
"M 177.0"	M 177.0	BOOL	// FLANCO NEGATIVO ( - ) - ALARMA No. 7
"M 177.1"	M 177.1	BOOL	// MARCA AUXILIAR - ALARMA No. 7
"M 177.2"	M 177.2	BOOL	// MARCA AUXILIAR - RECONOCIMIENTO DE ALARMA No. 7
"M 177.3"	M 177.3	BOOL	// MARCA AUXILIAR - RESTABLECIMIENTO DE ALARMA No. 7
"M 177.4"	M 177.4	BOOL	// MARCA AUXILIAR - INDICACION DE ALARMA No. 7
"M 177.5"	M 177.5	BOOL
"M 177.6"	M 177.6	BOOL
"M 177.7"	M 177.7	BOOL
"M 178.0"	M 178.0	BOOL	// FLANCO NEGATIVO ( - ) - ALARMA No. 8
"M 178.1"	M 178.1	BOOL	// MARCA AUXILIAR - ALARMA No. 8
"M 178.2"	M 178.2	BOOL	// MARCA AUXILIAR - RECONOCIMIENTO DE ALARMA No. 8
"M 178.3"	M 178.3	BOOL	// MARCA AUXILIAR - RESTABLECIMIENTO DE ALARMA No. 8
"M 178.4"	M 178.4	BOOL	// MARCA AUXILIAR - INDICACION DE ALARMA No. 8
"M 178.5"	M 178.5	BOOL
"M 178.6"	M 178.6	BOOL
"M 178.7"	M 178.7	BOOL
"M 179.0"	M 179.0	BOOL
"M 179.1"	M 179.1	BOOL
"M 179.2"	M 179.2	BOOL
"M 179.3"	M 179.3	BOOL
"M 179.4"	M 179.4	BOOL
"M 179.5"	M 179.5	BOOL
"M 179.6"	M 179.6	BOOL
"M 179.7"	M 179.7	BOOL
"M 180.0"	M 180.0	BOOL	// ALARMA No. 9
"M 180.1"	M 180.1	BOOL	// ALARMA No. 10
"M 180.2"	M 180.2	BOOL	// ALARMA No. 11
"M 180.3"	M 180.3	BOOL	// ALARMA No. 12
"M 180.4"	M 180.4	BOOL	// ALARMA No. 13
"M 180.5"	M 180.5	BOOL	// ALARMA No. 14
"M 180.6"	M 180.6	BOOL	// ALARMA No. 15
"M 180.7"	M 180.7	BOOL	// ALARMA No. 16
"M 181.0"	M 181.0	BOOL	// FLANCO POSITIVO ( + ) - ALARMA No. 9
"M 181.1"	M 181.1	BOOL	// MARCA AUXILIAR - ALARMA No. 9
"M 181.2"	M 181.2	BOOL	// MARCA AUXILIAR - RECONOCIMIENTO DE ALARMA No. 9
"M 181.3"	M 181.3	BOOL	// MARCA AUXILIAR - RESTABLECIMIENTO DE ALARMA No. 9
"M 181.4"	M 181.4	BOOL	// MARCA AUXILIAR - INDICACION DE ALARMA No. 9
"M 181.5"	M 181.5	BOOL
"M 181.6"	M 181.6	BOOL
"M 181.7"	M 181.7	BOOL
"M 182.0"	M 182.0	BOOL	// FLANCO POSITIVO ( + ) - ALARMA No. 10
"M 182.1"	M 182.1	BOOL	// MARCA AUXILIAR - ALARMA No. 10
"M 182.2"	M 182.2	BOOL	// MARCA AUXILIAR - RECONOCIMIENTO DE ALARMA No. 10
"M 182.3"	M 182.3	BOOL	// MARCA AUXILIAR - RESTABLECIMIENTO DE ALARMA No. 10
"M 182.4"	M 182.4	BOOL	// MARCA AUXILIAR - INDICACION DE ALARMA No. 10
"M 182.5"	M 182.5	BOOL
"M 182.6"	M 182.6	BOOL
"M 182.7"	M 182.7	BOOL
"M 183.0"	M 183.0	BOOL	// FLANCO POSITIVO ( + ) - ALARMA No. 11
"M 183.1"	M 183.1	BOOL	// MARCA AUXILIAR - ALARMA No. 11
"M 183.2"	M 183.2	BOOL	// MARCA AUXILIAR - RECONOCIMIENTO DE ALARMA No. 11
"M 183.3"	M 183.3	BOOL	// MARCA AUXILIAR - RESTABLECIMIENTO DE ALARMA No. 11
"M 183.4"	M 183.4	BOOL	// MARCA AUXILIAR - INDICACION DE ALARMA No. 11
"M 183.5"	M 183.5	BOOL
"M 183.6"	M 183.6	BOOL
"M 183.7"	M 183.7	BOOL
"M 184.0"	M 184.0	BOOL	// FLANCO POSITIVO ( + ) - ALARMA No. 12
"M 184.1"	M 184.1	BOOL	// MARCA AUXILIAR - ALARMA No. 12
"M 184.2"	M 184.2	BOOL	// MARCA AUXILIAR - RECONOCIMIENTO DE ALARMA No. 12
"M 184.3"	M 184.3	BOOL	// MARCA AUXILIAR - RESTABLECIMIENTO DE ALARMA No. 12
"M 184.4"	M 184.4	BOOL	// MARCA AUXILIAR - INDICACION DE ALARMA No. 12
"M 184.5"	M 184.5	BOOL
"M 184.6"	M 184.6	BOOL
"M 184.7"	M 184.7	BOOL
"M 185.0"	M 185.0	BOOL	// FLANCO POSITIVO ( + ) - ALARMA No. 13
"M 185.1"	M 185.1	BOOL	// MARCA AUXILIAR - ALARMA No. 13
"M 185.2"	M 185.2	BOOL	// MARCA AUXILIAR - RECONOCIMIENTO DE ALARMA No. 13
"M 185.3"	M 185.3	BOOL	// MARCA AUXILIAR - RESTABLECIMIENTO DE ALARMA No. 13
"M 185.4"	M 185.4	BOOL	// MARCA AUXILIAR - INDICACION DE ALARMA No. 13
"M 185.5"	M 185.5	BOOL
"M 185.6"	M 185.6	BOOL
"M 185.7"	M 185.7	BOOL
"M 186.0"	M 186.0	BOOL	// FLANCO POSITIVO ( + ) - ALARMA No. 14
"M 186.1"	M 186.1	BOOL	// MARCA AUXILIAR - ALARMA No. 14
"M 186.2"	M 186.2	BOOL	// MARCA AUXILIAR - RECONOCIMIENTO DE ALARMA No. 14
"M 186.3"	M 186.3	BOOL	// MARCA AUXILIAR - RESTABLECIMIENTO DE ALARMA No. 14
"M 186.4"	M 186.4	BOOL	// MARCA AUXILIAR - INDICACION DE ALARMA No. 14
"M 186.5"	M 186.5	BOOL
"M 186.6"	M 186.6	BOOL
"M 186.7"	M 186.7	BOOL
"M 187.0"	M 187.0	BOOL	// FLANCO POSITIVO ( + ) - ALARMA No. 15
"M 187.1"	M 187.1	BOOL	// MARCA AUXILIAR - ALARMA No. 15
"M 187.2"	M 187.2	BOOL	// MARCA AUXILIAR - RECONOCIMIENTO DE ALARMA No. 15
"M 187.3"	M 187.3	BOOL	// MARCA AUXILIAR - RESTABLECIMIENTO DE ALARMA No. 15
"M 187.4"	M 187.4	BOOL	// MARCA AUXILIAR - INDICACION DE ALARMA No. 15
"M 187.5"	M 187.5	BOOL
"M 187.6"	M 187.6	BOOL
"M 187.7"	M 187.7	BOOL
"M 188.0"	M 188.0	BOOL	// FLANCO POSITIVO ( + ) - ALARMA No. 16
"M 188.1"	M 188.1	BOOL	// MARCA AUXILIAR - ALARMA No. 16
"M 188.2"	M 188.2	BOOL	// MARCA AUXILIAR - RECONOCIMIENTO DE ALARMA No. 16
"M 188.3"	M 188.3	BOOL	// MARCA AUXILIAR - RESTABLECIMIENTO DE ALARMA No. 16
"M 188.4"	M 188.4	BOOL	// MARCA AUXILIAR - INDICACION DE ALARMA No. 16
"M 188.5"	M 188.5	BOOL
"M 188.6"	M 188.6	BOOL
"M 188.7"	M 188.7	BOOL
"M 189.0"	M 189.0	BOOL
"M 189.1"	M 189.1	BOOL
"M 189.2"	M 189.2	BOOL
"M 189.3"	M 189.3	BOOL
"M 189.4"	M 189.4	BOOL
"M 189.5"	M 189.5	BOOL
"M 189.6"	M 189.6	BOOL
"M 189.7"	M 189.7	BOOL
"M 190.0"	M 190.0	BOOL
"M 190.1"	M 190.1	BOOL	// BOTON DE RECONOCIMIENTO
"M 190.2"	M 190.2	BOOL	// BOTON DE RESTABLECIMIENTO
"M 190.3"	M 190.3	BOOL	// BOTON DE PRUEBA DE LAMPARAS
"M 190.4"	M 190.4	BOOL
"M 190.5"	M 190.5	BOOL
"M 190.6"	M 190.6	BOOL
"M 190.7"	M 190.7	BOOL
"M 191.0"	M 191.0	BOOL
"M 191.1"	M 191.1	BOOL
"M 191.2"	M 191.2	BOOL
"M 191.3"	M 191.3	BOOL
"M 191.4"	M 191.4	BOOL
"M 191.5"	M 191.5	BOOL
"M 191.6"	M 191.6	BOOL
"M 191.7"	M 191.7	BOOL
"M 192.0"	M 192.0	BOOL
"M 192.1"	M 192.1	BOOL
"M 192.2"	M 192.2	BOOL
"M 192.3"	M 192.3	BOOL
"M 192.4"	M 192.4	BOOL
"M 192.5"	M 192.5	BOOL
"M 192.6"	M 192.6	BOOL
"M 192.7"	M 192.7	BOOL
"M 193.0"	M 193.0	BOOL
"M 193.1"	M 193.1	BOOL
"M 193.2"	M 193.2	BOOL
"M 193.3"	M 193.3	BOOL
"M 193.4"	M 193.4	BOOL
"M 193.5"	M 193.5	BOOL
"M 193.6"	M 193.6	BOOL
"M 193.7"	M 193.7	BOOL
"M 194.0"	M 194.0	BOOL
"M 194.1"	M 194.1	BOOL
"M 194.2"	M 194.2	BOOL
"M 194.3"	M 194.3	BOOL
"M 194.4"	M 194.4	BOOL
"M 194.5"	M 194.5	BOOL
"M 194.6"	M 194.6	BOOL
"M 194.7"	M 194.7	BOOL
"M 195.0"	M 195.0	BOOL
"M 195.1"	M 195.1	BOOL
"M 195.2"	M 195.2	BOOL
"M 195.3"	M 195.3	BOOL
"M 195.4"	M 195.4	BOOL
"M 195.5"	M 195.5	BOOL
"M 195.6"	M 195.6	BOOL
"M 195.7"	M 195.7	BOOL
"M 196.0"	M 196.0	BOOL
"M 196.1"	M 196.1	BOOL
"M 196.2"	M 196.2	BOOL
"M 196.3"	M 196.3	BOOL
"M 196.4"	M 196.4	BOOL
"M 196.5"	M 196.5	BOOL
"M 196.6"	M 196.6	BOOL
"M 196.7"	M 196.7	BOOL
"M 197.0"	M 197.0	BOOL
"M 197.1"	M 197.1	BOOL
"M 197.2"	M 197.2	BOOL
"M 197.3"	M 197.3	BOOL
"M 197.4"	M 197.4	BOOL
"M 197.5"	M 197.5	BOOL
"M 197.6"	M 197.6	BOOL
"M 197.7"	M 197.7	BOOL
"M 198.0"	M 198.0	BOOL
"M 198.1"	M 198.1	BOOL
"M 198.2"	M 198.2	BOOL
"M 198.3"	M 198.3	BOOL
"M 198.4"	M 198.4	BOOL
"M 198.5"	M 198.5	BOOL
"M 198.6"	M 198.6	BOOL
"M 198.7"	M 198.7	BOOL
"M 199.0"	M 199.0	BOOL	// CYCLE_CLOCK MEMORY - 100 ms
"M 199.1"	M 199.1	BOOL	// CYCLE_CLOCK MEMORY - 200 ms
"M 199.2"	M 199.2	BOOL	// CYCLE_CLOCK MEMORY - 400 ms
"M 199.3"	M 199.3	BOOL	// CYCLE_CLOCK MEMORY - 500 ms
"M 199.4"	M 199.4	BOOL	// CYCLE_CLOCK MEMORY - 800 ms
"M 199.5"	M 199.5	BOOL	// CYCLE_CLOCK MEMORY - 1 seg
"M 199.6"	M 199.6	BOOL	// CYCLE_CLOCK MEMORY - 1.6 seg
"M 199.7"	M 199.7	BOOL	// CYCLE_CLOCK MEMORY - 2 seg
"."	M 255.7	BOOL	// DUMMY
"M405.0"	M 405.0	BOOL	// EVENTO # 1 / PRESENTE
"M 405.1"	M 405.1	BOOL	// FLANCO POSITIVO EVENTO # 1
"M 408.0"	M 408.0	BOOL	// INDICACION DE ALARMA
"M 410.4"	M 410.4	BOOL	// BOTON DE RESTABLECIMENTO
"M410.5"	M 410.5	BOOL	// BOTON DE RECONOCIMENTO
"M410.6"	M 410.6	BOOL	// PRUEBA DE LAMAPARAS
"20S4"	M 410.7	BOOL	// BOTON DE SILENCIAR BOCINA
"MB 0"	MB 0	BYTE
"MB 1"	MB 1	BYTE
"MB 2"	MB 2	BYTE
"MB 3"	MB 3	BYTE
"MB 4"	MB 4	BYTE
"MB 5"	MB 5	BYTE
"MB 6"	MB 6	BYTE
"MB 7"	MB 7	BYTE
"MB 8"	MB 8	BYTE
"MB 9"	MB 9	BYTE
"MB 10"	MB 10	BYTE
"MB 11"	MB 11	BYTE
"MB 12"	MB 12	BYTE
"MB 13"	MB 13	BYTE
"MB 14"	MB 14	BYTE
"MB 15"	MB 15	BYTE
"MB 16"	MB 16	BYTE
"MB 17"	MB 17	BYTE
"MB 18"	MB 18	BYTE
"MB 19"	MB 19	BYTE
"MB 20"	MB 20	BYTE
"MB 21"	MB 21	BYTE
"MB 22"	MB 22	BYTE
"MB 23"	MB 23	BYTE
"MB 24"	MB 24	BYTE
"MB 25"	MB 25	BYTE
"MB 26"	MB 26	BYTE
"MB 27"	MB 27	BYTE
"MB 28"	MB 28	BYTE
"MB 29"	MB 29	BYTE
"MB 30"	MB 30	BYTE
"MB 31"	MB 31	BYTE
"MB 32"	MB 32	BYTE
"MB 33"	MB 33	BYTE
"MB 34"	MB 34	BYTE
"MB 35"	MB 35	BYTE
"MB 36"	MB 36	BYTE
"MB 37"	MB 37	BYTE
"MB 38"	MB 38	BYTE
"MB 39"	MB 39	BYTE
"MB 40"	MB 40	BYTE
"MB 41"	MB 41	BYTE
"MB 42"	MB 42	BYTE
"MB 43"	MB 43	BYTE
"MB 44"	MB 44	BYTE
"MB 45"	MB 45	BYTE
"MB 46"	MB 46	BYTE
"MB 47"	MB 47	BYTE
"MB 48"	MB 48	BYTE
"MB 49"	MB 49	BYTE
"MB 50"	MB 50	BYTE
"MB 51"	MB 51	BYTE
"MB 52"	MB 52	BYTE
"MB 53"	MB 53	BYTE
"MB 54"	MB 54	BYTE
"MB 55"	MB 55	BYTE
"MB 56"	MB 56	BYTE
"MB 57"	MB 57	BYTE
"MB 58"	MB 58	BYTE
"MB 59"	MB 59	BYTE
"MB 60"	MB 60	BYTE
"MB 61"	MB 61	BYTE
"MB 62"	MB 62	BYTE
"MB 63"	MB 63	BYTE
"MB 64"	MB 64	BYTE
"MB 65"	MB 65	BYTE
"MB 66"	MB 66	BYTE
"MB 67"	MB 67	BYTE
"MB 68"	MB 68	BYTE
"MB 69"	MB 69	BYTE
"MB 70"	MB 70	BYTE
"MB 71"	MB 71	BYTE
"MB 72"	MB 72	BYTE
"MB 73"	MB 73	BYTE
"MB 74"	MB 74	BYTE
"MB 75"	MB 75	BYTE
"MB 76"	MB 76	BYTE
"MB 77"	MB 77	BYTE
"MB 78"	MB 78	BYTE
"MB 79"	MB 79	BYTE
"MB 80"	MB 80	BYTE
"MB 81"	MB 81	BYTE
"MB 82"	MB 82	BYTE
"MB 83"	MB 83	BYTE
"MB 84"	MB 84	BYTE
"MB 85"	MB 85	BYTE
"MB 86"	MB 86	BYTE
"MB 87"	MB 87	BYTE
"MB 88"	MB 88	BYTE
"MB 89"	MB 89	BYTE
"MB 90"	MB 90	BYTE
"MB 91"	MB 91	BYTE
"MB 92"	MB 92	BYTE
"MB 93"	MB 93	BYTE
"MB 94"	MB 94	BYTE
"MB 95"	MB 95	BYTE
"MB 96"	MB 96	BYTE
"MB 97"	MB 97	BYTE
"MB 98"	MB 98	BYTE
"MB 99"	MB 99	BYTE
"MB 100"	MB 100	BYTE
"MB 101"	MB 101	BYTE
"MB 102"	MB 102	BYTE
"MB 103"	MB 103	BYTE
"MB 104"	MB 104	BYTE
"MB 105"	MB 105	BYTE
"MB 106"	MB 106	BYTE
"MB 107"	MB 107	BYTE
"MB 108"	MB 108	BYTE
"MB 109"	MB 109	BYTE
"MB 110"	MB 110	BYTE
"MB 111"	MB 111	BYTE
"MB 112"	MB 112	BYTE
"MB 113"	MB 113	BYTE
"MB 114"	MB 114	BYTE
"MB 115"	MB 115	BYTE
"MB 116"	MB 116	BYTE
"MB 117"	MB 117	BYTE
"MB 118"	MB 118	BYTE
"MB 119"	MB 119	BYTE
"MB 120"	MB 120	BYTE
"MB 121"	MB 121	BYTE
"MB 122"	MB 122	BYTE
"MB 123"	MB 123	BYTE
"MB 124"	MB 124	BYTE
"MB 125"	MB 125	BYTE
"MB 126"	MB 126	BYTE
"MB 127"	MB 127	BYTE
"MB 128"	MB 128	BYTE
"MB 129"	MB 129	BYTE
"MB 130"	MB 130	BYTE
"MB 131"	MB 131	BYTE
"MB 132"	MB 132	BYTE
"MB 133"	MB 133	BYTE
"MB 134"	MB 134	BYTE
"MB 135"	MB 135	BYTE
"MB 136"	MB 136	BYTE
"MB 137"	MB 137	BYTE
"MB 138"	MB 138	BYTE
"MB 139"	MB 139	BYTE
"MB 140"	MB 140	BYTE	// AJUSTE DE ALARMA - HORAS ( INDICACION )
"MB 141"	MB 141	BYTE	// AJUSTE DE ALARMA - MINUTOS ( INDICACION )
"MB 142"	MB 142	BYTE	// RELOJ DESPERTADOR - HORAS ( INDICACION )
"MB 143"	MB 143	BYTE	// RELOJ DESPERTADOR - MINUTOS ( INDICACION )
"MB 144"	MB 144	BYTE
"MB 145"	MB 145	BYTE
"MB 146"	MB 146	BYTE
"MB 147"	MB 147	BYTE
"MB 148"	MB 148	BYTE
"MB 149"	MB 149	BYTE
"MB 150"	MB 150	BYTE
"MB 151"	MB 151	BYTE
"MB 152"	MB 152	BYTE
"MB 153"	MB 153	BYTE
"MB 154"	MB 154	BYTE
"MB 155"	MB 155	BYTE
"MB 156"	MB 156	BYTE
"MB 157"	MB 157	BYTE
"MB 158"	MB 158	BYTE
"MB 159"	MB 159	BYTE
"MB 160"	MB 160	BYTE
"MB 161"	MB 161	BYTE	// AJUSTE DE ALARMA - MINUTOS ( INDICACION BCD )
"MB 162"	MB 162	BYTE
"MB 163"	MB 163	BYTE	// AJUSTE DE ALARMA - HORAS ( INDICACION BCD )
"MB 164"	MB 164	BYTE
"MB 165"	MB 165	BYTE
"MB 166"	MB 166	BYTE
"MB 167"	MB 167	BYTE	// RELOJ DESPERTADOR - MINUTOS ( INDICACION BCD )
"MB 168"	MB 168	BYTE
"MB 169"	MB 169	BYTE	// RELOJ DESPERTADOR - HORAS ( INDICACION BCD )
"MB 170"	MB 170	BYTE
"MB 171"	MB 171	BYTE
"MB 172"	MB 172	BYTE
"MB 173"	MB 173	BYTE
"MB 174"	MB 174	BYTE
"MB 175"	MB 175	BYTE
"MB 176"	MB 176	BYTE
"MB 177"	MB 177	BYTE
"MB 178"	MB 178	BYTE
"MB 179"	MB 179	BYTE
"MB 180"	MB 180	BYTE
"MB 181"	MB 181	BYTE
"MB 182"	MB 182	BYTE
"MB 183"	MB 183	BYTE
"MB 184"	MB 184	BYTE
"MB 185"	MB 185	BYTE
"MB 186"	MB 186	BYTE
"MB 187"	MB 187	BYTE
"MB 188"	MB 188	BYTE
"MB 189"	MB 189	BYTE
"MB 190"	MB 190	BYTE
"MB 191"	MB 191	BYTE
"MB 192"	MB 192	BYTE
"MB 193"	MB 193	BYTE
"MB 194"	MB 194	BYTE
"MB 195"	MB 195	BYTE
"MB 196"	MB 196	BYTE
"MB 197"	MB 197	BYTE
"MB 198"	MB 198	BYTE
"MB 199"	MB 199	BYTE
"MW 30"	MW 30	WORD	// INDICACION DE TIEMPO - LUZ ROJA ( BCD )
"MW 32"	MW 32	WORD	// INDICACION DE TIEMPO - LUZ VERDE ( BCD )
"MW 34"	MW 34	WORD	// INDICACION DE TIEMPO - LUZ AMARILLA ( BCD )
"MW 36"	MW 36	WORD	// INDICACION DE TIEMPO - FLECHA_LUZ VERDE
"MW 50"	MW 50	WORD	// INDICACION DE TIEMPO ( LUZ ROJA - BCD )
"MW 52"	MW 52	WORD	// INIDICACION DE TIEMPO ( LUZ VERDE - BCD )
"MW 54"	MW 54	WORD	// VALOR DE AJUSTE DEL CONTADOR
"MW 56"	MW 56	WORD	// INDICACION DE CONTADOR
"MW 58"	MW 58	WORD	// INDICADOR DE CONTADOR DE PULSOS
"MW 60"	MW 60	WORD
"MW 62"	MW 62	WORD
"MW 64"	MW 64	WORD
"MW 66"	MW 66	WORD
"MW 120"	MW 120	WORD	// INIDICACION DE TIEMPO ( LUZ ROJA - BCD ) - INICIO
"MW 122"	MW 122	WORD	// INIDICACION DE TIEMPO ( LUZ ROJA - BCD )
"MW 124"	MW 124	WORD	// INIDICACION DE TIEMPO ( LUZ VERDE - BCD )
"MW 126"	MW 126	WORD	// INIDICACION DE TIEMPO ( LUZ AMARILLA - BCD )
"MW 128"	MW 128	WORD	// INIDICACION DE TIEMPO ( FLECHA - LUZ VERDE - BCD )
"MW 140"	MW 140	WORD	// INIDICACION DE TIEMPO ( LUZ ROJA - ENTERO ) - INICIO
"MW 142"	MW 142	WORD	// INIDICACION DE TIEMPO ( LUZ ROJA - ENTERO )
"MW 144"	MW 144	WORD	// INIDICACION DE TIEMPO ( LUZ VERDE - ENTERO )
"MW 146"	MW 146	WORD	// INIDICACION DE TIEMPO ( LUZ AMARILLA - ENTERO )
"MW 148"	MW 148	INT	// INIDICACION DE TIEMPO ( FLECHA - LUZ VERDE - ENTERO )
"MW 150"	MW 150	INT	// INDICACION DE MINUTOS ( ALARMA - ENTERO )
"MW 152"	MW 152	INT	// INDICACION DE HORAS ( ALARMA - ENTERO )
"MW 154"	MW 154	INT	// INDICACION DE SEGUNDOS ( RELOJ - ENTERO )
"MW 156"	MW 156	INT	// INDICACION DE MINUTOS ( RELOJ - ENTERO )
"MW 158"	MW 158	INT	// INDICACION DE HORAS ( RELOJ - ENTERO )
"MW 160"	MW 160	WORD	// INDICACION DE MINUTOS ( ALARMA - BCD )
"MW 162"	MW 162	WORD	// INDICACION DE HORAS ( ALARMA - BCD )
"MW 164"	MW 164	WORD	// INDICACION DE SEGUNDOS ( RELOJ - BCD )
"MW 166"	MW 166	WORD	// INDICACION DE MINUTOS ( RELOJ - BCD )
"MW 168"	MW 168	WORD	// INDICACION DE HORAS ( RELOJ - BCD )
"CYCL_EXC"	OB 1	OB 1	// Cycle Execution
"CYC_INT5"	OB 35	OB 35	// Cyclic Interrupt 5
"CYCL_FLT"	OB 80	OB 80	// Cycle Time Fault
"I/O_FLT1"	OB 82	OB 82	// I/O Point Fault 1
"I/O_FLT2"	OB 83	OB 83	// I/O Point Fault 2
"OBNL_FLT"	OB 85	OB 85	// OB Not Loaded Fault
"RACK_FLT"	OB 86	OB 86	// Loss of Rack Fault
"COMM_FLT"	OB 87	OB 87	// Communication Fault
"COMPLETE RESTART"	OB 100	OB 100	// Complete Restart
"PROG_ERR"	OB 121	OB 121	// Programming Error
"MOD_ERR"	OB 122	OB 122	// Module Access Error
"1H1"	Q 0.0	BOOL	// LAMPARA INDICADORA # 1
"2H1"	Q 0.1	BOOL	// LAMPARA INDICADORA # 2
"3H1"	Q 0.2	BOOL	// LAMPARA INDICADORA # 3
"4H1"	Q 0.3	BOOL	// LAMPARA INDICADORA # 4
"5H1"	Q 0.4	BOOL	// LAMPARA INDICADORA # 5
"6H1"	Q 0.5	BOOL	// LAMPARA INDICADORA # 6
"7H1"	Q 0.6	BOOL	// LAMPARA INDICADORA # 7
"8H1"	Q 0.7	BOOL	// LAMPARA INDICADORA # 8
"1H2"	Q 1.0	BOOL	// LAMPARA INDICADORA # 9
"2H2"	Q 1.1	BOOL	// LAMPARA INDICADORA # 10
"3H2"	Q 1.2	BOOL	// LAMPARA INDICADORA # 11
"4H2"	Q 1.3	BOOL	// LAMPARA INDICADORA # 12
"5H2"	Q 1.4	BOOL	// LAMPARA INDICADORA # 13
"6H2"	Q 1.5	BOOL	// LAMPARA INDICADORA # 14
"7H2"	Q 1.6	BOOL	// LAMPARA INDICADORA # 15
"8H2"	Q 1.7	BOOL	// LAMPARA INDICADORA # 16
"1H3"	Q 2.0	BOOL	// LAMPARA INDICADORA # 17
"2H3"	Q 2.1	BOOL	// LAMPARA INDICADORA # 18
"3H3"	Q 2.2	BOOL	// LAMPARA INDICADORA # 19
"4H3"	Q 2.3	BOOL	// LAMPARA INDICADORA # 20
"5H3"	Q 2.4	BOOL	// LAMPARA INDICADORA # 21
"6H3"	Q 2.5	BOOL	// LAMPARA INDICADORA # 22
"7H3"	Q 2.6	BOOL	// LAMPARA INDICADORA # 23
"8H3"	Q 2.7	BOOL	// LAMPARA INDICADORA # 24
"1H4"	Q 3.0	BOOL	// LAMPARA INDICADORA # 25
"2H4"	Q 3.1	BOOL	// LAMPARA INDICADORA # 26
"3H4"	Q 3.2	BOOL	// LAMPARA INDICADORA # 27
"4H4"	Q 3.3	BOOL	// LAMPARA INDICADORA # 28
"5H4"	Q 3.4	BOOL	// LAMPARA INDICADORA # 29
"6H4"	Q 3.5	BOOL	// LAMPARA INDICADORA # 30
"7H4"	Q 3.6	BOOL	// LAMPARA INDICADORA # 31
"8H4"	Q 3.7	BOOL	// LAMPARA INDICADORA # 32
"5KM1"	Q 4.0	BOOL	// CONTACTOR PRINCIPAL 5KM1
"5KM2"	Q 4.1	BOOL	// CONTACTOR PRINCIPAL 5KM2
"5KM3"	Q 4.2	BOOL	// CONTACTOR PRINCIPAL 5KM3
"5KM4"	Q 4.3	BOOL	// CONTACTOR PRINCIPAL 5KM4
"A 4.4"	Q 4.4	BOOL
"A 4.5"	Q 4.5	BOOL
"A 4.6"	Q 4.6	BOOL
"A 4.7"	Q 4.7	BOOL
"6KM1"	Q 5.0	BOOL	// CONTACTOR PRINCIPAL 6KM1
"6KM2"	Q 5.1	BOOL	// CONTACTOR PRINCIPAL 6KM2
"6KM3"	Q 5.2	BOOL	// CONTACTOR PRINCIPAL 6KM3
"A 5.3"	Q 5.3	BOOL
"A 5.4"	Q 5.4	BOOL
"A 5.5"	Q 5.5	BOOL
"A 5.6"	Q 5.6	BOOL
"A 5.7"	Q 5.7	BOOL
"1KM1"	Q 6.0	BOOL	// CONTACTOR PRINCIPAL 1KM1
"2KM1."	Q 6.1	BOOL	// CONTACTOR PRINCIPAL 2KM1
"2KM2."	Q 6.2	BOOL	// CONTACTOR PRINCIPAL 2KM2
"A 6.3"	Q 6.3	BOOL
"A 6.4"	Q 6.4	BOOL
"2KM1"	Q 6.5	BOOL	// CONTACTOR PRINCIPAL 2KM1
"2KM2"	Q 6.6	BOOL	// CONTACTOR PRINCIPAL 2KM2
"A 6.7"	Q 6.7	BOOL
"A 8.0"	Q 8.0	BOOL
"H1"	Q 8.1	BOOL	// TRANSPORTADOR - LUZ INDICADORA L_BAY1
"H2"	Q 8.2	BOOL	// TRANSPORTADOR - LUZ INDICADORA L_BAY2
"H3"	Q 8.3	BOOL	// TRANSPORTADOR - LUZ INDICADORA L_BAY3
"H4"	Q 8.4	BOOL	// TRANSPORTADOR - LUZ INDICADORA L_BAY-LB
"K_CONV_RIGTH"	Q 8.5	BOOL	// TRANSPORTADOR - DESPLAZAMIENTO A LA DERECHA
"K_CONV_LEFT"	Q 8.6	BOOL	// TRANSPORTADOR - DESPLAZAMIENTO A LA IZQUIERDA
"HORN"	Q 8.7	BOOL	// TRANSPORTADOR - BOCINA
"3KM1"	Q 12.0	BOOL	// CONTACTOR PRINCIPAL 3KM1
"3KM2"	Q 12.1	BOOL	// CONTACTOR PRINCIPAL 3KM2
"A 12.2"	Q 12.2	BOOL
"A 12.3"	Q 12.3	BOOL
"A 12.4"	Q 12.4	BOOL
"A 12.5"	Q 12.5	BOOL
"A 12.6"	Q 12.6	BOOL
"A 12.7"	Q 12.7	BOOL
"4KM1"	Q 13.0	BOOL	// CONTACTOR PRINCIPAL 4KM1
"4KM2"	Q 13.1	BOOL	// CONTACTOR PRINCIPAL 4KM2
"4KM3"	Q 13.2	BOOL	// CONTACTOR PRINCIPAL 4KM3
"A 13.3"	Q 13.3	BOOL
"A 13.4"	Q 13.4	BOOL
"A 13.5"	Q 13.5	BOOL
"A 13.6"	Q 13.6	BOOL
"A 13.7"	Q 13.7	BOOL
"A 14.0"	Q 14.0	BOOL
"A 14.1"	Q 14.1	BOOL
"A 14.2"	Q 14.2	BOOL
"A 14.3"	Q 14.3	BOOL
"A 14.4"	Q 14.4	BOOL
"A 14.5"	Q 14.5	BOOL
"A 14.6"	Q 14.6	BOOL
"A 14.7"	Q 14.7	BOOL
"A 15.0"	Q 15.0	BOOL
"A 15.1"	Q 15.1	BOOL
"A 15.2"	Q 15.2	BOOL
"A 15.3"	Q 15.3	BOOL
"A 15.4"	Q 15.4	BOOL
"A 15.5"	Q 15.5	BOOL
"A 15.6"	Q 15.6	BOOL
"A 15.7"	Q 15.7	BOOL
"7KM1"	Q 16.0	BOOL	// CONTACTOR DE VELOCIDAD LENTA
"7KM2"	Q 16.1	BOOL	// CONTACTOR DE VELOCIDAD RAPIDA
"7KM3"	Q 16.2	BOOL	// CONTACTOR DE VELOCIDAD RAPIDA
"A16.3"	Q 16.3	BOOL
"A16.4"	Q 16.4	BOOL
"A16.5"	Q 16.5	BOOL
"7KM10"	Q 17.0	BOOL	// CONTACTOR DE BAJADA
"7KM20"	Q 17.1	BOOL	// CONTACTOR DE SUBIDA
"7H1."	Q 21.0	BOOL
"7H2."	Q 21.1	BOOL
"7H3."	Q 21.2	BOOL
"1H1A"	Q 124.0	BOOL	// INDICACION DE OPERACION LOCAL # 1
"1H1B"	Q 124.1	BOOL	// INDICACION DE OPERACION REMOTA # 1
"2H1A"	Q 124.2	BOOL	// INDICACION DE OPERACION LOCAL # 2
"2H1B"	Q 124.3	BOOL	// INDICACION DE OPERACION REMOTA # 2
"3H1A"	Q 124.4	BOOL	// INDICACION DE OPERACION LOCAL # 3
"3H1B"	Q 124.5	BOOL	// INDICACION DE OPERACION REMOTA # 3
"4H1A"	Q 124.6	BOOL	// INDICACION DE OPERACION LOCAL # 4
"4H1B"	Q 124.7	BOOL	// INDICACION DE OPERACION REMOTA # 4
"5H1A"	Q 125.0	BOOL	// INDICACION DE OPERACION LOCAL # 5
"5H1B"	Q 125.1	BOOL	// INDICACION DE OPERACION REMOTA # 5
"6H1A"	Q 125.2	BOOL	// INDICACION DE OPERACION LOCAL # 6
"6H1B"	Q 125.3	BOOL	// INDICACION DE OPERACION REMOTA # 6
"7H1A"	Q 125.4	BOOL	// INDICACION DE OPERACION LOCAL # 7
"7H1B"	Q 125.5	BOOL	// INDICACION DE OPERACION REMOTA # 7
"8H1A"	Q 125.6	BOOL	// INDICACION DE OPERACION LOCAL # 8
"8H1B"	Q 125.7	BOOL	// INDICACION DE OPERACION REMOTA # 8
"RDREC"	SFB 52	SFB 52	// Read a Process Data Record
"RALRM"	SFB 54	SFB 54	// Receive Alarm Data
"ALARM_SQ"	SFC 17	SFC 17	// Generate Block-Related Messages with Acknowledgment
"ALARM_S"	SFC 18	SFC 18	// Generate Permanently Acknowledged Block-Related Messages
"WR_USMSG"	SFC 52	SFC 52	// Write a User-Defined Diagnostic Event to the Diagnostic Buffer
"TIME_TCK"	SFC 64	SFC 64	// Read the System Time
"T 1"	T 1	TIMER
"KT2"	T 2	TIMER	// TIEMPO DE CONMUTACION - CIRCUITO DE TEMPORIZACION
"T 3"	T 3	TIMER
"T 4"	T 4	TIMER
"KT5"	T 5	TIMER	// TIEMPO DE TRANSFERENCIA ( ESTRELLA - DELTA )
"T 6"	T 6	TIMER
"7KT4"	T 7	TIMER	// TIEMPO DE SUPERVISION - CONMUTACION DE VELOCIDADES
"T 8"	T 8	TIMER
"T 9"	T 9	TIMER
"T 10"	T 10	TIMER	// GENERADOR DE IMPULSOS ( PARTE I )
"T 11"	T 11	TIMER	// GENERADOR DE IMPULSOS ( PARTE II )
"T 12"	T 12	TIMER	// TIEMPO DE DURACION ( LUZ ROJA )
"T 13"	T 13	TIMER	// TIEMPO DE DURACION ( LUZ VERDE )
"T 14"	T 14	TIMER	// TIEMPO DE DURACION ( LUZ AMARILLA )
"T 15"	T 15	TIMER	// TIEMPO DE DURACION ( FLECHA - LUZ VERDE )
"T 16"	T 16	TIMER
"T 17"	T 17	TIMER
"T 18"	T 18	TIMER
"T 19"	T 19	TIMER
"T 20"	T 20	TIMER	// TIEMPO DE SUPERVISION DE CONMUTACION ESTRELLA - DELTA
"T 21"	T 21	TIMER
"T 22"	T 22	TIMER
"T 23"	T 23	TIMER
"T 24"	T 24	TIMER
"T 25"	T 25	TIMER
"T 26"	T 26	TIMER
"T 27"	T 27	TIMER
"T 28"	T 28	TIMER
"T 29"	T 29	TIMER
"T 30"	T 30	TIMER
"T 31"	T 31	TIMER
"T 32"	T 32	TIMER
"T 33"	T 33	TIMER
"T 34"	T 34	TIMER
"T 35"	T 35	TIMER
"T 36"	T 36	TIMER
"T 37"	T 37	TIMER
"T 38"	T 38	TIMER
"T 39"	T 39	TIMER
"T 40"	T 40	TIMER	// GENERADOR DE IMPULSOS ( PARTE I )
"T 41"	T 41	TIMER	// TIEMPO DE DURACION / INICIO ( LUZ ROJA )
"T 42"	T 42	TIMER	// TIEMPO DE DURACION ( LUZ ROJA )
"T 43"	T 43	TIMER	// TIEMPO DE DURACION ( LUZ VERDE )
"T 44"	T 44	TIMER	// TIEMPO DE DURACION ( LUZ AMARILLA )
"T 45"	T 45	TIMER	// TIEMPO DE DURACION ( FLECHA - LUZ VERDE )
"T 46"	T 46	TIMER
"T 47"	T 47	TIMER
"T 48"	T 48	TIMER
"T 49"	T 49	TIMER
"T 50"	T 50	TIMER
"T 51"	T 51	TIMER
"T 52"	T 52	TIMER
"T 53"	T 53	TIMER
"T 54"	T 54	TIMER
"T 55"	T 55	TIMER
"T 56"	T 56	TIMER
"T 57"	T 57	TIMER
"T 58"	T 58	TIMER
"T 59"	T 59	TIMER
"T 60"	T 60	TIMER
"T 61"	T 61	TIMER
"T 62"	T 62	TIMER
"T 63"	T 63	TIMER
"T 64"	T 64	TIMER
"T 65"	T 65	TIMER
"T 66"	T 66	TIMER
"T 67"	T 67	TIMER
"T 68"	T 68	TIMER
"T 69"	T 69	TIMER
"T 70"	T 70	TIMER
"T 71"	T 71	TIMER
"T 72"	T 72	TIMER
"T 73"	T 73	TIMER
"T 74"	T 74	TIMER
"T 75"	T 75	TIMER
"T 76"	T 76	TIMER
"T 77"	T 77	TIMER
"T 78"	T 78	TIMER
"T 79"	T 79	TIMER
"T 80"	T 80	TIMER
"T 81"	T 81	TIMER
"T 82"	T 82	TIMER
"T 83"	T 83	TIMER
"T 84"	T 84	TIMER
"T 85"	T 85	TIMER
"T 86"	T 86	TIMER
"T 87"	T 87	TIMER
"T 88"	T 88	TIMER
"T 89"	T 89	TIMER
"T 90"	T 90	TIMER
"T 91"	T 91	TIMER
"T 92"	T 92	TIMER
"T 93"	T 93	TIMER
"T 94"	T 94	TIMER
"T 95"	T 95	TIMER
"T 96"	T 96	TIMER
"T 97"	T 97	TIMER
"T 98"	T 98	TIMER
"T 99"	T 99	TIMER
"T 100"	T 100	TIMER	// TIEMPO DE REINICIO DE BOCINA
"T 101"	T 101	TIMER
"T 102"	T 102	TIMER
"T 103"	T 103	TIMER
"T 104"	T 104	TIMER
"T 105"	T 105	TIMER
"T 106"	T 106	TIMER
"T 107"	T 107	TIMER
"T 108"	T 108	TIMER
"T 109"	T 109	TIMER
"T 110"	T 110	TIMER
"T 111"	T 111	TIMER
"T 112"	T 112	TIMER
"T 113"	T 113	TIMER
"T 114"	T 114	TIMER
"T 115"	T 115	TIMER
"T 116"	T 116	TIMER
"T 117"	T 117	TIMER
"T 118"	T 118	TIMER
"T 119"	T 119	TIMER	// TIEMPO DE SUPERVISION DE FRECUENCIA
"T 120"	T 120	TIMER	// TEMPORIZADOR DE IMPULSO
"T 121"	T 121	TIMER	// TEMPORIZADOR DE IMPULSO EXTENDIDO
"T 122"	T 122	TIMER	// TEMPORIZADOR DE RETARDO A LA CONEXION
"T 123"	T 123	TIMER	// TEMPORIZADOR RETARDO A LA DESCONEXION - RETENTIVO
"T 124"	T 124	TIMER	// TEMPORIZADOR - RETARDO A LA DESCONEXION
"T 126"	T 126	TIMER
"T 127"	T 127	TIMER	// GENERADOR DE IMPULSOS
"T 128"	T 128	TIMER
"T 129"	T 129	TIMER
"T 130"	T 130	TIMER
"T 131"	T 131	TIMER
"T 132"	T 132	TIMER
"T 133"	T 133	TIMER
"T 134"	T 134	TIMER
"T 135"	T 135	TIMER
"T 136"	T 136	TIMER
"T 137"	T 137	TIMER
"T 138"	T 138	TIMER
"T 139"	T 139	TIMER
"T 140"	T 140	TIMER
"T 141"	T 141	TIMER
"T 142"	T 142	TIMER
"T 143"	T 143	TIMER
"T 144"	T 144	TIMER
"T 145"	T 145	TIMER
"T 146"	T 146	TIMER
"T 147"	T 147	TIMER
"T 148"	T 148	TIMER
"T 149"	T 149	TIMER
"T 150"	T 150	TIMER
"T 151"	T 151	TIMER
"T 152"	T 152	TIMER
"T 153"	T 153	TIMER
"T 154"	T 154	TIMER
"T 155"	T 155	TIMER
"T 156"	T 156	TIMER
"T 157"	T 157	TIMER
"T 158"	T 158	TIMER
"T 159"	T 159	TIMER
"T 160"	T 160	TIMER
"T 161"	T 161	TIMER
"T 162"	T 162	TIMER
"T 163"	T 163	TIMER
"T 164"	T 164	TIMER
"T 165"	T 165	TIMER
"T 166"	T 166	TIMER
"T 167"	T 167	TIMER
"T 168"	T 168	TIMER
"T 169"	T 169	TIMER
"T 170"	T 170	TIMER
"T 171"	T 171	TIMER
"T 172"	T 172	TIMER
"T 173"	T 173	TIMER
"T 174"	T 174	TIMER
"T 175"	T 175	TIMER
"T 176"	T 176	TIMER
"T 177"	T 177	TIMER
"T 178"	T 178	TIMER
"T 179"	T 179	TIMER
"T 180"	T 180	TIMER
"T 181"	T 181	TIMER
"T 182"	T 182	TIMER
"T 183"	T 183	TIMER
"T 184"	T 184	TIMER
"T 185"	T 185	TIMER
"T 186"	T 186	TIMER
"T 187"	T 187	TIMER
"T 188"	T 188	TIMER
"T 189"	T 189	TIMER
"T 190"	T 190	TIMER
"T 191"	T 191	TIMER
"T 192"	T 192	TIMER
"T 193"	T 193	TIMER
"T 194"	T 194	TIMER
"T 195"	T 195	TIMER
"T 196"	T 196	TIMER
"T 197"	T 197	TIMER
"T 198"	T 198	TIMER
"T 199"	T 199	TIMER
"T 200"	T 200	TIMER
"T 201"	T 201	TIMER
"T 202"	T 202	TIMER
"T 203"	T 203	TIMER
"T 204"	T 204	TIMER
"T 205"	T 205	TIMER
"T 206"	T 206	TIMER
"T 207"	T 207	TIMER
"T 208"	T 208	TIMER
"T 209"	T 209	TIMER
"T 210"	T 210	TIMER
"T 211"	T 211	TIMER
"T 212"	T 212	TIMER
"T 213"	T 213	TIMER
"T 214"	T 214	TIMER
"T 215"	T 215	TIMER
"T 216"	T 216	TIMER
"T 217"	T 217	TIMER
"T 218"	T 218	TIMER
"T 219"	T 219	TIMER
"T 220"	T 220	TIMER
"T 221"	T 221	TIMER
"T 222"	T 222	TIMER
"T 223"	T 223	TIMER
"T 224"	T 224	TIMER
"T 225"	T 225	TIMER
"T 226"	T 226	TIMER
"T 227"	T 227	TIMER
"T 228"	T 228	TIMER
"T 229"	T 229	TIMER
"T 230"	T 230	TIMER
"T 231"	T 231	TIMER
"T 232"	T 232	TIMER
"T 233"	T 233	TIMER
"T 234"	T 234	TIMER
"T 235"	T 235	TIMER
"T 236"	T 236	TIMER
"T 237"	T 237	TIMER
"T 238"	T 238	TIMER
"T 239"	T 239	TIMER
"T 240"	T 240	TIMER
"T 241"	T 241	TIMER
"T 242"	T 242	TIMER
"T 243"	T 243	TIMER
"T 244"	T 244	TIMER
"T 245"	T 245	TIMER
"T 246"	T 246	TIMER
"T 247"	T 247	TIMER
"T 248"	T 248	TIMER
"T 249"	T 249	TIMER
"T 250"	T 250	TIMER
"T 251"	T 251	TIMER
"T 252"	T 252	TIMER
"T 253"	T 253	TIMER
"T 254"	T 254	TIMER
"T 255"	T 255	TIMER
"T 256"	T 256	TIMER
"ENTRADA_000"	VAT 1	
"ENTRADA_004"	VAT 2	
"ENTRADA_006"	VAT 3	
"ENTRADA_008"	VAT 4	
"ENTRADA_012"	VAT 5	
"ENTRADA_016"	VAT 6	
"ENTRADA_124"	VAT 7	
"SALIDA_000"	VAT 8	
"SALIDA_004"	VAT 9	
"SALIDA_006"	VAT 10	
"SALIDA_008"	VAT 11	
"SALIDA_012"	VAT 12	
"SALIDA_016"	VAT 13	
"SALIDA_124"	VAT 14	
"EJERCICIO # 1"	VAT 15		// CIRCUITO DE ENCLAVAMIENTO
"ent0"	VAT 16		// CIRCUITO DE TEMPORIZACION
"ent1"	VAT 17	
"ent2"	VAT 18		// entrada2
"ent4"	VAT 19		// Modulo E 4
"ent5"	VAT 20		// Modulo E 5
"ent6"	VAT 21		// Modulo E6
"ent8"	VAT 22		// Modulo E8
"ent12"	VAT 23		// Modulo E12
"ent13"	VAT 24		// Modulo E13
"ent16"	VAT 25		// Modulo entrada 20
"ent17"	VAT 26		// Modulo E17
"sal0"	VAT 27		// Modulo S0
"sal1"	VAT 28	
"sal2"	VAT 29		// Modulo salida 2
END_SYMBOL_TABLE

// FB 126: know-how protected block, not included

// FB 127: know-how protected block, not included

FUNCTION "TE-M/V" : VOID	// FC 10
AUTHOR : SIMATIC
FAMILY : EA_DIS
NAME : TE_M_V
VERSION : 3.0
BEGIN
// (block stored without names or comments; labels and parameter names are numbered)
NETWORK
TITLE =
      L     0;
      L     #PARAM19;
      ==I;
      JC    M001;
      T     MW 212;
      L     MB 212;
      T     LW 10;
      OPN   DB [LW 10];
      L     MB 213;
      SLW   3;
      LAR1;
      L     DBW [AR1,P#0.0];
      L     MB 212;
      T     LW 10;
      OPN   DB [LW 10];
      L     MB 213;
      SLW   3;
      LAR1;
      L     DBW [AR1,P#0.0];
M001: T     MB 211;
      OPN   #PARAM16;
      L     #PARAM17;
      T     MW 212;
      L     MB 213;
      SLW   3;
      LAR1;
      L     DBW [AR1,P#0.0];
      T     MW 200;
      L     DBW [AR1,P#2.0];
      T     MW 202;
      L     DBW [AR1,P#4.0];
      T     MW 204;
      L     0;
      T     MW 206;
      A     #PARAM1;
      =     M 206.7;
      A     #PARAM2;
      =     M 203.0;
      A     #PARAM3;
      AN    M 202.2;
      =     M 210.7;
      A     #PARAM3;
      =     M 202.2;
      A     #PARAM4;
      AN    #PARAM7;
      AN    M 200.0;
      =     M 210.6;
      A     #PARAM4;
      AN    #PARAM7;
      =     M 200.0;
      A     #PARAM7;
      AN    #PARAM4;
      AN    M 200.1;
      =     M 210.4;
      A     #PARAM7;
      AN    #PARAM4;
      =     M 200.1;
      A     #PARAM8;
      AN    M 202.3;
      =     M 210.5;
      A     #PARAM8;
      =     M 202.3;
      A     #PARAM9;
      =     M 200.7;
      A     #PARAM10;
      =     M 206.4;
      A     #PARAM6;
      =     M 206.5;
      A     #PARAM5;
      =     M 206.6;
      A     #PARAM11;
      =     M 206.3;
      A     #PARAM12;
      =     M 206.1;
      A     #PARAM13;
      =     M 206.0;
      A     #PARAM14;
      =     M 200.4;
NETWORK
TITLE =
      A     M 206.1;
      AN    M 206.0;
      =     M 201.3;
      A     M 206.0;
      AN    M 206.1;
      =     M 201.5;
NETWORK
TITLE =
      A     M 211.2;
      A     M 211.1;
      AN    M 202.0;
      AN    M 200.1;
      =     M 210.3;
      A     M 211.2;
      A     M 211.1;
      =     M 202.0;
      A     M 211.3;
      A     M 211.1;
      AN    M 202.1;
      AN    M 200.0;
      =     M 210.2;
      A     M 211.3;
      A     M 211.1;
      =     M 202.1;
NETWORK
TITLE =
      A     M 210.5;
      A     M 206.5;
      AN    M 202.2;
      O;
      A     M 210.2;
      AN    M 211.2;
      A(;
      AN    M 202.2;
      ON    M 206.5;
      );
      O;
      A     M 210.4;
      AN    M 200.0;
      A(;
      AN    M 202.2;
      ON    M 206.5;
      );
      A(;
      AN    M 211.2;
      ON    M 211.1;
      );
      =     M 207.2;
NETWORK
TITLE =
      A     M 210.7;
      A     M 206.5;
      O;
      A     M 210.3;
      A(;
      AN    M 202.3;
      ON    M 206.5;
      );
      O;
      A     M 210.6;
      A(;
      AN    M 202.3;
      ON    M 206.5;
      );
      A(;
      AN    M 211.3;
      ON    M 211.1;
      );
      =     M 207.3;
NETWORK
TITLE =
      A     M 211.3;
      AN    M 203.6;
      O     M 210.5;
      =     M 207.4;
      A     M 211.3;
      =     M 203.6;
      A     M 211.2;
      AN    M 203.5;
      O     M 210.7;
      =     M 207.5;
      A     M 211.2;
      =     M 203.5;
NETWORK
TITLE =
      A     M 202.3;
      A     M 206.5;
      O;
      A     M 211.3;
      A     M 211.1;
      O     M 200.1;
      =     M 207.6;
      A     M 202.2;
      A     M 206.5;
      O;
      A     M 211.2;
      A     M 211.1;
      O     M 200.0;
      =     M 207.7;
      A     M 207.6;
      ON    M 203.0;
      O     M 206.4;
      A     M 207.7;
      O;
      A(;
      A     M 207.7;
      ON    M 200.7;
      O     M 206.7;
      A     M 207.6;
      );
      O;
      A     M 206.7;
      A     M 206.4;
      =     M 201.1;
NETWORK
TITLE =
      L     MB 205;
      T     MB 209;
      L     0;
      >I;
      JC    M004;
      AN    M 206.7;
      ON    M 203.7;
      JC    M002;
      L     #PARAM15;
      T     MB 204;
      L     6;
      JU    M003;
M002: A     M 201.5;
      L     5;
      JC    M003;
      AN    M 201.3;
      L     1;
      JC    M004;
M003: T     MB 209;
M004: NOP   0;
NETWORK
TITLE =
      L     MB 205;
      L     1;
      <>I;
      JC    M007;
      A     M 206.7;
      JC    M007;
      A     M 207.4;
      A     M 200.1;
      O     M 207.2;
      A     M 200.7;
      A     M 201.3;
      O     M 206.4;
      JC    M005;
      A     M 201.5;
      L     4;
      JC    M006;
      JU    M007;
M005: L     #PARAM15;
      T     MB 204;
      L     2;
M006: T     MB 209;
M007: NOP   0;
NETWORK
TITLE =
      L     MB 205;
      L     2;
      <>I;
      JC    M009;
      A     M 207.3;
      A     M 203.0;
      AN    M 206.4;
      O     M 206.7;
      L     6;
      L     #PARAM15;
      JC    M008;
      A     M 201.5;
      L     5;
      L     0;
      JC    M008;
      L     MB 204;
      >=I;
      L     3;
      L     0;
      JC    M008;
      AN    "M 1.3";
      JC    M009;
      L     MB 204;
      +     -1;
      T     MB 204;
      JU    M009;
M008: T     MB 204;
      TAK;
      T     MB 209;
M009: NOP   0;
NETWORK
TITLE =
      L     MB 205;
      L     3;
      <>I;
      JC    M012;
      AN    M 206.7;
      ON    M 203.7;
      JC    M010;
      L     #PARAM15;
      T     MB 204;
      L     6;
      JC    M011;
M010: A     M 207.5;
      A     M 201.3;
      L     1;
      JC    M011;
      AN    M 207.4;
      ON    M 201.5;
      JC    M012;
      L     5;
M011: T     MB 209;
M012: NOP   0;
NETWORK
TITLE =
      L     MB 205;
      L     4;
      <>I;
      JC    M015;
      AN    M 206.7;
      ON    M 203.7;
      JC    M013;
      L     #PARAM15;
      T     MB 204;
      L     6;
      JC    M014;
M013: A     M 207.5;
      A     M 201.3;
      L     1;
      JC    M014;
      ON    M 207.4;
      ON    M 201.5;
      JC    M015;
      L     5;
M014: T     MB 209;
M015: NOP   0;
NETWORK
TITLE =
      L     MB 205;
      L     5;
      <>I;
      JC    M018;
      L     6;
      A     M 207.5;
      A     M 200.0;
      O     M 207.3;
      A     M 203.0;
      AN    M 206.4;
      O     M 206.7;
      JC    M016;
      AN    M 201.3;
      AN    M 200.4;
      JC    M018;
      L     8;
      JU    M017;
M016: L     #PARAM15;
      T     MB 204;
      TAK;
M017: T     MB 209;
M018: NOP   0;
NETWORK
TITLE =
      L     MB 205;
      L     6;
      <>I;
      JC    M020;
      A     M 207.2;
      A     M 200.7;
      O     M 206.4;
      AN    M 206.7;
      L     2;
      L     #PARAM15;
      JC    M019;
      A     M 201.3;
      A     M 203.7;
      A     M 206.7;
      L     9;
      L     0;
      JC    M019;
      A     M 201.3;
      L     1;
      L     0;
      JC    M019;
      L     MB 204;
      >=I;
      L     7;
      L     0;
      JC    M019;
      AN    "M 1.3";
      JC    M020;
      L     MB 204;
      +     -1;
      T     MB 204;
      JU    M020;
M019: T     MB 204;
      TAK;
      T     MB 209;
M020: NOP   0;
NETWORK
TITLE =
      L     MB 205;
      L     7;
      <>I;
      JC    M022;
      A     M 207.5;
      A     M 201.3;
      L     1;
      JC    M021;
      AN    M 207.4;
      ON    M 201.5;
      JC    M022;
      L     5;
M021: T     MB 209;
M022: NOP   0;
NETWORK
TITLE =
      L     MB 205;
      L     8;
      <>I;
      JC    M025;
      AN    M 206.7;
      ON    M 203.7;
      JC    M023;
      L     #PARAM15;
      T     MB 204;
      L     6;
      JC    M024;
M023: A     M 207.5;
      A     M 201.3;
      AN    M 200.4;
      L     1;
      JC    M024;
      ON    M 207.4;
      ON    M 201.5;
      JC    M025;
      L     5;
M024: T     MB 209;
M025: NOP   0;
NETWORK
TITLE =
      L     MB 205;
      L     9;
      <>I;
      JC    M028;
      A     M 207.5;
      A     M 200.1;
      A     M 200.7;
      O     M 206.4;
      AN    M 206.7;
      L     2;
      JC    M026;
      AN    M 207.5;
      JC    M028;
      L     1;
      JU    M027;
M026: L     #PARAM15;
      T     MB 204;
      TAK;
M027: T     MB 209;
M028: NOP   0;
NETWORK
TITLE =
      L     MB 209;
      T     MB 205;
      L     9;
      <=I;
      JC    M029;
      L     0;
      T     MW 204;
M029: NOP   0;
NETWORK
TITLE =
      AN    M 201.3;
      AN    M 201.5;
      =     M 206.2;
      A     M 209.0;
      ON    M 209.1;
      A     M 206.2;
      =     M 200.6;
      A     M 209.2;
      O     M 209.3;
      AN    M 209.0;
      AN    M 209.1;
      AN    M 206.2;
      =     M 200.5;
      A     M 209.0;
      A     M 209.1;
      A     M 209.2;
      AN    M 206.2;
      =     M 200.2;
      A     M 209.0;
      A     M 209.1;
      AN    M 209.2;
      AN    M 206.2;
      =     M 200.3;
      AN    M 209.0;
      A     M 209.1;
      A     M 207.6;
      AN    M 200.1;
      =     M 201.7;
      AN    M 209.0;
      A     M 209.1;
      A     M 207.7;
      AN    M 207.3;
      =     M 201.6;
NETWORK
TITLE =
      A     M 201.1;
      =     M 203.3;
      A     M 209.0;
      A     M 209.3;
      O     M 200.4;
      O     M 200.5;
      O     M 200.3;
      O     M 200.2;
      =     M 201.0;
      AN    M 209.0;
      AN    M 209.1;
      A     M 209.2;
      AN    M 206.2;
      O;
      A     M 209.0;
      A     M 209.1;
      A     M 209.2;
      AN    M 206.2;
      =     M 202.4;
      AN    M 209.0;
      A     M 209.1;
      A     M 209.2;
      =     M 202.6;
      A     M 202.4;
      O     M 202.6;
      =     M 201.2;
      A     M 209.0;
      A     M 209.1;
      AN    M 209.2;
      O     M 209.3;
      AN    M 206.2;
      =     M 202.5;
      AN    M 209.0;
      A     M 209.1;
      AN    M 209.2;
      =     M 202.7;
      A     M 202.5;
      O     M 202.7;
      =     M 201.4;
      AN    M 201.4;
      A     M 206.0;
      =     M 203.2;
      AN    M 201.2;
      A     M 206.1;
      =     M 203.1;
NETWORK
TITLE =
      A     M 201.0;
      O     M 203.3;
      =     #PARAM23;
      A     M 201.3;
      =     #PARAM21;
      A     M 201.5;
      =     #PARAM22;
      A     M 201.0;
      A     "M 1.6";
      O     M 203.3;
      O     #PARAM11;
      =     #PARAM26;
      A     M 202.7;
      A     "M 0.5";
      O;
      A     M 202.5;
      A     "M 1.6";
      O     M 203.2;
      O     #PARAM11;
      =     #PARAM25;
      A     M 202.6;
      A     "M 0.5";
      O;
      A     M 202.4;
      A     "M 1.6";
      O     M 203.1;
      O     #PARAM11;
      =     #PARAM24;
NETWORK
TITLE =
      A(;
      AN    M 206.6;
      A     M 209.0;
      AN    M 209.1;
      A     M 209.2;
      O;
      A     M 209.1;
      AN    M 209.2;
      );
      AN    M 200.6;
      AN    M 200.3;
      =     #PARAM28;
      A(;
      A     M 209.0;
      AN    M 209.1;
      AN    M 209.2;
      AN    M 206.6;
      O;
      A     M 209.1;
      A     M 209.2;
      );
      AN    M 200.6;
      AN    M 200.2;
      =     #PARAM27;
      L     MW 200;
      T     DBW [AR1,P#0.0];
      L     MW 202;
      T     DBW [AR1,P#2.0];
      L     MW 204;
      T     DBW [AR1,P#4.0];
      L     MW 206;
      T     DBW [AR1,P#6.0];
      L     0;
      L     #PARAM20;
      ==I;
      JC    M032;
      T     MW 206;
      T     MW 220;
      L     MB 206;
      SLW   3;
      LAR1;
      L     DBW [AR1,P#2.0];
      T     MW 208;
      L     MW 220;
      SLW   12;
      SRW   12;
      T     MW 220;
      L     8;
      L     MB 221;
      >I;
      JC    M030;
      +     -8;
      SLW   8;
      INC   208;
      JU    M031;
M030: SLW   8;
      INC   209;
M031: T     MW 210;
      L     MB 210;
      L     MB 211;
      SLW   3;
      OW;
      LAR2;
      A     M 201.0;
      O     M 203.3;
      =     M [AR2,P#0.0];
      L     MB 206;
      SLW   3;
      LAR1;
      L     MW 208;
      T     DBW [AR1,P#2.0];
M032: L     0;
      L     #PARAM18;
      ==I;
      BEC;
      T     MW 212;
      L     MB 212;
      T     LW 10;
      OPN   DB [LW 10];
      L     MB 213;
      SLW   3;
      LAR1;
      L     MW 200;
      T     DBW [AR1,P#0.0];
      L     MW 202;
      T     DBW [AR1,P#2.0];
END_FUNCTION

